// TIA Portal V21 program export: 5 tag tables, 1 data types, 6 data blocks, 4 code blocks (in call order from the OBs), 2 instance data blocks

VAR_GLOBAL   // PLC tag table "A0.300"
   tESTE_01 AT %I15.0 : Bool;
END_VAR

VAR_GLOBAL   // PLC tag table "Cabinet_Config"
   M_Power_line_3_4_Available AT %M100.0 : Bool;
   M_Power_line_5_6_Available AT %M100.1 : Bool;
   M_Safety_zone_3_4_Available AT %M101.0 : Bool;
   M_Safety_zone_5_6_Available AT %M101.1 : Bool;
   M_Safety_zone_7_8_Available AT %M101.2 : Bool;
   M_Fast_doors_Enabled AT %M102.0 : Bool;
   M_Wrapping_machine_Enabled AT %M102.1 : Bool;
   M_CabinetNumberOutOfRange AT %M110.0 : Bool;
   M_HWCombiNumberOutOfRange AT %M110.1 : Bool;
END_VAR
VAR_GLOBAL CONSTANT   // user constants
   K_MaxCabinetNumber : UInt := 10;   // Max. number of C0 cabinets allowed
   K_MaxHWCombiNumber : UInt := 16;   // Max. number of defined PLC hardware combinations
END_VAR

VAR_GLOBAL   // PLC tag table "Cabinet_Management"
   M_Power_cabinet AT %M2.0 : Bool;
   M_Power_L1 AT %M3.0 : Bool;
   M_Power_L2 AT %M3.1 : Bool;
   M_Power_L3 AT %M3.2 : Bool;
   M_Power_L4 AT %M3.3 : Bool;
   M_Power_L5 AT %M3.4 : Bool;
   M_Power_L6 AT %M3.5 : Bool;
   M_Buzzer AT %M4.0 : Bool;
   M_NF_Cabinet_fault AT %M5.0 : Bool;
   M_Cabinet_fault AT %M5.1 : Bool;
   M_Rearm_Power_Cabinet AT %M6.0 : Bool;
   M_Reset_safety_Z1 AT %M7.0 : Bool;
   M_Reset_safety_Z2 AT %M7.1 : Bool;
   M_Reset_safety_Z3 AT %M7.2 : Bool;
   M_Reset_safety_Z4 AT %M7.3 : Bool;
   M_Reset_safety_Z5 AT %M7.4 : Bool;
   M_Reset_safety_Z6 AT %M7.5 : Bool;
   M_Reset_safety_Z7 AT %M7.6 : Bool;
   M_Reset_safety_Z8 AT %M7.7 : Bool;
   M_Facility_OK AT %M6.7 : Bool;   // Conveyors status OK
END_VAR

VAR_GLOBAL   // PLC tag table "Default tag table"
   System_Byte AT %MB1 : Byte;
   FirstScan AT %M1.0 : Bool;
   DiagStatusUpdate AT %M1.1 : Bool;
   AlwaysTRUE AT %M1.2 : Bool;
   AlwaysFALSE AT %M1.3 : Bool;
   Clock_Byte AT %MB0 : Byte;
   Clock_10Hz AT %M0.0 : Bool;
   Clock_5Hz AT %M0.1 : Bool;
   "Clock_2.5Hz" AT %M0.2 : Bool;
   Clock_2Hz AT %M0.3 : Bool;
   "Clock_1.25Hz" AT %M0.4 : Bool;
   Clock_1Hz AT %M0.5 : Bool;
   "Clock_0.625Hz" AT %M0.6 : Bool;
   "Clock_0.5Hz" AT %M0.7 : Bool;
   "+C0_K0.001" AT %I0.0 : Bool;   // Phase monitor OK
   "+C0_AUX/OK" AT %I0.1 : Bool;   // Auxiliary services protection OK
   "+C0_CAL/OK" AT %I0.2 : Bool;   // Heater protection OK
   "+C0_PE/OK" AT %I0.3 : Bool;   // Insulation monitor OK
   "+C0_Spare_101.4" AT %I0.4 : Bool;   // Spare
   "+C0_Spare_101.5" AT %I0.5 : Bool;   // Spare
   "+C0_Spare_101.6" AT %I0.6 : Bool;   // Spare
   "+C0_Spare_101.7" AT %I0.7 : Bool;   // Spare
   "+C0_S2.101" AT %I1.0 : Bool;   // Cabinet reset (power lines + emergencies)
   "+C0_S2.001" AT %I1.1 : Bool;   // Cabinet power lines deactivation
   "+C0_S2.002" AT %I1.2 : Bool;   // Acoustic warning stop
   "+C0_Spare_102.3" AT %I1.3 : Bool;   // Spare
   "+C0_IF5" AT %I1.4 : Bool;   // External machine interface 5
   "+C0_IF6" AT %I1.5 : Bool;   // External machine interface 6
   "+C0_IF7" AT %I1.6 : Bool;   // External machine interface 7
   "+C0_IF8" AT %I1.7 : Bool;   // External machine interface 8
   "+C0_F2.101" AT %I2.0 : Bool;   // 400V Power L1 protection OK
   "+C0_Q1.001" AT %I2.1 : Bool;   // Power L1 is active
   "+C0_1SE1" AT %I2.2 : Bool;   // Emergency stop 1 Z1 OK
   "+C0_1SE2" AT %I2.3 : Bool;   // Emergency stop 2 Z1 OK
   "+C0_F2.102" AT %I2.4 : Bool;   // 400V Power L2 protection OK
   "+C0_Q1.002" AT %I2.5 : Bool;   // Power L2 is active
   "+C0_2SE1" AT %I2.6 : Bool;   // Emergency stop 1 Z2 OK
   "+C0_2SE2" AT %I2.7 : Bool;   // Emergency stop 2 Z2 OK
   "+C0_F2.103" AT %I3.0 : Bool;   // 400V Power L3 protection OK
   "+C0_Q1.003" AT %I3.1 : Bool;   // Power L3 is active
   "+C0_3SE1" AT %I3.2 : Bool;   // Emergency stop 1 Z3 OK
   "+C0_3SE2" AT %I3.3 : Bool;   // Emergency stop 2 Z3 OK
   "+C0_F2.104" AT %I3.4 : Bool;   // 400V Power L4 protection OK
   "+C0_Q1.004" AT %I3.5 : Bool;   // Power L4 is active
   "+C0_4SE1" AT %I3.6 : Bool;   // Emergency stop 1 Z4 OK
   "+C0_4SE2" AT %I3.7 : Bool;   // Emergency stop 2 Z4 OK
   "+C0_F2.105" AT %I4.0 : Bool;   // 400V Power L5 protection OK
   "+C0_Q1.005" AT %I4.1 : Bool;   // Power L5 is active
   "+C0_5SE1" AT %I4.2 : Bool;   // Emergency stop 1 Z5 OK
   "+C0_5SE2" AT %I4.3 : Bool;   // Emergency stop 2 Z5 OK
   "+C0_F2.106" AT %I4.4 : Bool;   // 400V Power L6 protection OK
   "+C0_Q1.006" AT %I4.5 : Bool;   // Power L6 is active
   "+C0_6SE1" AT %I4.6 : Bool;   // Emergency stop 1 Z6 OK
   "+C0_6SE2" AT %I4.7 : Bool;   // Emergency stop 2 Z6 OK
   "+C0_Spare_106.1" AT %I5.1 : Bool;   // Spare
   "+C0_7SE1" AT %I5.2 : Bool;   // Emergency stop 1 Z7 OK
   "+C0_7SE2" AT %I5.3 : Bool;   // Emergency stop 2 Z7 OK
   "+C0_Spare_106.4" AT %I5.4 : Bool;   // Spare
   "+C0_Spare_106.5" AT %I5.5 : Bool;   // Spare
   "+C0_8SE1" AT %I5.6 : Bool;   // Emergency stop 1 Z8 OK
   "+C0_8SE2" AT %I5.7 : Bool;   // Emergency stop 2 Z8 OK
   "+C0_F0.199 -F2.199" AT %I6.0 : Bool;   // Wrapping machine protection OK
   "+C0_ENF1" AT %I6.1 : Bool;   // Wrapping machine is ready
   "+C0_ENF2" AT %I6.2 : Bool;   // Wrapping machine entry consent
   "+C0_ENF3" AT %I6.3 : Bool;   // Wrapping machine completed process
   "+C0_Spare_107.4" AT %I6.4 : Bool;   // Spare
   "+C0_Spare_107.5" AT %I6.5 : Bool;   // Spare
   "+C0_Spare_107.6" AT %I6.6 : Bool;   // Spare
   "+C0_Spare_107.7" AT %I6.7 : Bool;   // Spare
   "+C0_F0.190+" AT %I7.0 : Bool;   // Fast doors protection OK
   "+C0_1PR1" AT %I7.1 : Bool;   // Fast door 1 is open
   "+C0_1PR2" AT %I7.2 : Bool;   // Fast door 1 is closed
   "+C0_2PR1" AT %I7.3 : Bool;   // Fast door 2 is open
   "+C0_2PR2" AT %I7.4 : Bool;   // Fast door 2 is closed
   "+C0_3PR1" AT %I7.5 : Bool;   // Fast door 3 is open
   "+C0_3PR2" AT %I7.6 : Bool;   // Fast door 3 is closed
   "+C0_Spare_108.7" AT %I7.7 : Bool;   // Spare
   "+C0_Buzzer" AT %Q0.0 : Bool;   // Beacon buzzer
   "+C0_Beacon_Green" AT %Q0.1 : Bool;   // Beacon green lamp
   "+C0_Beacon_Red" AT %Q0.2 : Bool;   // Beacon red lamp
   "+C0_Spare_151.3" AT %Q0.3 : Bool;   // Spare
   "+C0_PEM" AT %Q0.4 : Bool;   // Cabinet emergency stop is active
   "+C0_RE" AT %Q0.5 : Bool;   // Cabinet power lines are active
   "+C0_Spare_151.6" AT %Q0.6 : Bool;   // Spare
   "+C0_Spare_151.7" AT %Q0.7 : Bool;   // Spare
   "+C0_K1.007" AT %Q1.0 : Bool;   // External machine interface 1
   "+C0_K1.008" AT %Q1.1 : Bool;   // External machine interface 2
   "+C0_K1.009" AT %Q1.2 : Bool;   // External machine interface 3
   "+C0_K1.010" AT %Q1.3 : Bool;   // External machine interface 4
   "+C0_Spare_152.4" AT %Q1.4 : Bool;   // Spare
   "+C0_Spare_152.5" AT %Q1.5 : Bool;   // Spare
   "+C0_Spare_152.6" AT %Q1.6 : Bool;   // Spare
   "+C0_Spare_152.7" AT %Q1.7 : Bool;   // Spare
   "+C0_K1.001" AT %Q2.0 : Bool;   // 400V Power L1 activation
   "+C0_K1.002" AT %Q2.1 : Bool;   // 400V Power L2 activation
   "+C0_K1.003" AT %Q2.2 : Bool;   // 400V Power L3 activation
   "+C0_K1.004" AT %Q2.3 : Bool;   // 400V Power L4 activation
   "+C0_K1.005" AT %Q2.4 : Bool;   // 400V Power L5 activation
   "+C0_K1.006" AT %Q2.5 : Bool;   // 400V Power L6 activation
   "+C0_Spare_153.6" AT %Q2.6 : Bool;   // Spare
   "+C0_Spare_153.7" AT %Q2.7 : Bool;   // Spare
   "+C0_K1.020" AT %Q3.0 : Bool;   // Wrapping machine exit request
   "+C0_Spare_154.1" AT %Q3.1 : Bool;   // Spare
   "+C0_K1.030" AT %Q3.2 : Bool;   // Open fast door 1
   "+C0_K1.031" AT %Q3.3 : Bool;   // Close fast door 1
   "+C0_K1.032" AT %Q3.4 : Bool;   // Open fast door 2
   "+C0_K1.033" AT %Q3.5 : Bool;   // Close fast door 2
   "+C0_K1.035" AT %Q3.7 : Bool;   // Close fast door 3
   "+C0_S1.001_1" AT %I100.0 : Bool;   // Cabinet emergency stop ch1
   "+C0_Spare_201.1" AT %I100.1 : Bool;   // Spare
   "+C0_Spare_201.2" AT %I100.2 : Bool;   // Spare
   "+C0_Spare_201.3" AT %I100.3 : Bool;   // Spare
   "+C0_S1.001_2" AT %I100.4 : Bool;   // Cabinet emergency stop ch2
   "+C0_Spare_201.5" AT %I100.5 : Bool;   // Spare
   "+C0_Spare_201.6" AT %I100.6 : Bool;   // Spare
   "+C0_Spare_201.7" AT %I100.7 : Bool;   // Spare
   "+C0_1EM1" AT %I107.0 : Bool;   // Emergency stop Z1 ch1
   "+C0_2EM1" AT %I107.1 : Bool;   // Emergency stop Z2 ch1
   "+C0_K4.011-111-012-112" AT %I107.2 : Bool;   // Safety Z1 relays feedback
   "+C0_Spare_202.3" AT %I107.3 : Bool;   // Spare
   "+C0_1EM2" AT %I107.4 : Bool;   // Emergency stop Z1 ch2
   "+C0_2EM2" AT %I107.5 : Bool;   // Emergency stop Z2 ch2
   "+C0_K4.021-121-022-122" AT %I107.6 : Bool;   // Safety Z2 relays feedback
   "+C0_Spare_202.7" AT %I107.7 : Bool;   // Sapre
   "+C0_3EM1" AT %I114.0 : Bool;   // Emergency stop Z3 ch1
   "+C0_4EM1" AT %I114.1 : Bool;   // Emergency stop Z4 ch1
   "+C0_K4.031-131-032-132" AT %I114.2 : Bool;   // Safety Z3 relays feedback
   "+C0_Spare_203.3" AT %I114.3 : Bool;   // Spare
   "+C0_3EM2" AT %I114.4 : Bool;   // Emergency stop Z3 ch2
   "+C0_4EM2" AT %I114.5 : Bool;   // Emergency stop Z4 ch2
   "+C0_K4.041-141-042-142" AT %I114.6 : Bool;   // Safety Z4 relays feedback
   "+C0_Spare_203.7" AT %I114.7 : Bool;   // Spare
   "+C0_5EM1" AT %I121.0 : Bool;   // Emergency stop Z5 ch1
   "+C0_6EM1" AT %I121.1 : Bool;   // Emergency stop Z6 ch1
   "+C0_K4.051-151-052-152" AT %I121.2 : Bool;   // Safety Z5 relays feedback
   "+C0_Spare_204.3" AT %I121.3 : Bool;   // Spare
   "+C0_5EM2" AT %I121.4 : Bool;   // Emergency stop Z5 ch2
   "+C0_6EM2" AT %I121.5 : Bool;   // Emergency stop Z6 ch2
   "+C0_K4.061-161-062-162" AT %I121.6 : Bool;   // Safety Z6 relays feedback
   "+C0_Spare_204.7" AT %I121.7 : Bool;   // Spare
   "+C0_7EM1" AT %I128.0 : Bool;   // Emergency stop Z7 ch1
   "+C0_8EM1" AT %I128.1 : Bool;   // Emergency stop Z8 ch1
   "+C0_K4.071-171-072-172" AT %I128.2 : Bool;   // Safety Z7 relays feedback
   "+C0_Spare_205.3" AT %I128.3 : Bool;   // Spare
   "+C0_7EM2" AT %I128.4 : Bool;   // Emergency stop Z7 ch2
   "+C0_8EM2" AT %I128.5 : Bool;   // Emergency stop Z8 ch2
   "+C0_K4.081-181-082-182" AT %I128.6 : Bool;   // Safety Z8 relays feedback
   "+C0_Spare_205.7" AT %I128.7 : Bool;   // Spare
   "+C0_K4.011-111" AT %Q200.0 : Bool;   // Safety Z1 ch1 relay activation
   "+C0_K4.012-112" AT %Q200.1 : Bool;   // Safety Z1 ch2 relay activation
   "+C0_K4.021-121" AT %Q200.2 : Bool;   // Safety Z2 ch1 relay activation
   "+C0_K4.022-122" AT %Q200.3 : Bool;   // Safety Z2 ch2 relay activation
   "+C0_K4.031-131" AT %Q200.4 : Bool;   // Safety Z3 ch1 relay activation
   "+C0_K4.032-132" AT %Q200.5 : Bool;   // Safety Z3 ch2 relay activation
   "+C0_K4.041-141" AT %Q200.6 : Bool;   // Safety Z4 ch1 relay activation
   "+C0_K4.042-142" AT %Q200.7 : Bool;   // Safety Z4 ch2 relay activation
   "+C0_K4.051-151" AT %Q206.0 : Bool;   // Safety Z5 ch1 relay activation
   "+C0_K4.052-152" AT %Q206.1 : Bool;   // Safety Z5 ch2 relay activation
   "+C0_K4.061-161" AT %Q206.2 : Bool;   // Safety Z6 ch1 relay activation
   "+C0_K4.062-162" AT %Q206.3 : Bool;   // Safety Z6 ch2 relay activation
   "+C0_K4.071-171" AT %Q206.4 : Bool;   // Safety Z7 ch1 relay activation
   "+C0_K4.072-172" AT %Q206.5 : Bool;   // Safety Z7 ch2 relay activation
   "+C0_K4.081-181" AT %Q206.6 : Bool;   // Safety Z8 ch1 relay activation
   "+C0_K4.082-182" AT %Q206.7 : Bool;   // Safety Z8 ch2 relay activation
   "+C0_A0.101" AT %IB0 : Byte;
   "+C0_A0.102" AT %IB1 : Byte;
   "+C0_A0.103" AT %IB2 : Byte;
   "+C0_A0.104" AT %IB3 : Byte;
   "+C0_A0.105" AT %IB4 : Byte;
   "+C0_A0.106" AT %IB5 : Byte;
   "+C0_A0.107" AT %IB6 : Byte;
   "+C0_A0.108" AT %IB7 : Byte;
   "+C0_Spare_106.0" AT %I5.0 : Bool;   // Spare
   "+C0_K1.034" AT %Q3.6 : Bool;   // Open fast door 3
   RONDI_PEM_20260514 AT %M650.0 : Bool;   // VARIABLE DE PUESTA EN MARCHA
END_VAR

VAR_GLOBAL   // PLC tag table "Process_Data"
   IB_Byte0 AT %IB400 : Byte;
   IB_Byte1 AT %IB401 : Byte;
   OB_Byte0 AT %QB400 : Byte;
   OB_Byte1 AT %QB401 : Byte;
   OB_Byte2 AT %QB402 : Byte;
   OB_Byte3 AT %QB403 : Byte;
   OB_Byte4 AT %QB404 : Byte;
   OB_Byte5 AT %QB405 : Byte;
   OB_Byte6 AT %QB406 : Byte;
   OB_Byte7 AT %QB407 : Byte;
   OB_Byte8 AT %QB408 : Byte;
   OB_Byte9 AT %QB409 : Byte;
   OB_Byte10 AT %QB410 : Byte;
   IB_Byte2 AT %IB402 : Byte;
   IB_Byte3 AT %IB403 : Byte;
   OB_Byte11 AT %QB411 : Byte;
END_VAR

TYPE "TypeC0"
   STRUCT
      Heated_Lines_Enabled : Bool;   // true = Heated line/s are enabled
      Insulation_Monitor_Enabled : Bool;   // true = Insulation monitor is enabled
      Power_L2_Disabled : Bool;   // true = Power L2 is disabled
      Power_L4_Disabled : Bool;   // true = Power L4 is disabled
      Power_L6_Disabled : Bool;   // true = Power L6 is disabled
      Safety_Z2_Disabled : Bool;   // true = Safety Z2 is disabled
      Safety_Z4_Disabled : Bool;   // true = Safety Z4 is disabled
      Safety_Z6_Disabled : Bool;   // true = Safety Z6 is disabled
      Safety_Z8_Disabled : Bool;   // true = Safety Z8 is disabled
      HWCombiNumber : Int;   // PLC hardware combination number
   END_STRUCT;
END_TYPE

DATA_BLOCK "HWData"   // DB3
{ S7_Optimized_Access := 'TRUE' }
// stored: AutoNumber false, MemoryReserve 0
   VAR
      CombiNumber : Int := 0;   // Number according to PLC hardware combination
      ConfigSlots : Array[1.."K_MaxHWCombiNumber"] of "LCC_typeCPUET200SP";   // Slots configurations for all PLC hardware combinations
      CPUET200SP_StatusID : USInt;
      CPUET200SP_Status : DWord;
      CPUET200SP_Config { S7_SetPoint := 'True'} : "LCC_typeCPUET200SP";   // Slots configuration for selected hardware combination
   END_VAR
BEGIN
   ConfigSlots[1].slots[4].actSlotNumber := 132;
   ConfigSlots[1].slots[5].actSlotNumber := 133;
   ConfigSlots[1].slots[6].actSlotNumber := 134;
   ConfigSlots[1].slots[7].actSlotNumber := 7;
   ConfigSlots[1].slots[8].actSlotNumber := 136;
   ConfigSlots[1].slots[9].actSlotNumber := 9;
   ConfigSlots[1].slots[10].actSlotNumber := 10;
   ConfigSlots[1].slots[11].actSlotNumber := 11;
   ConfigSlots[1].slots[12..16].actSlotNumber := 0;
   ConfigSlots[1].slots[17].actSlotNumber := 12;
   ConfigSlots[1].slots[18].actSlotNumber := 13;
   ConfigSlots[1].slots[19].actSlotNumber := 14;
   ConfigSlots[1].slots[20].actSlotNumber := 0;
   ConfigSlots[1].slots[21].actSlotNumber := 15;
   ConfigSlots[2].slots[4].actSlotNumber := 132;
   ConfigSlots[2].slots[5].actSlotNumber := 133;
   ConfigSlots[2].slots[6].actSlotNumber := 134;
   ConfigSlots[2].slots[7].actSlotNumber := 7;
   ConfigSlots[2].slots[8].actSlotNumber := 136;
   ConfigSlots[2].slots[9].actSlotNumber := 9;
   ConfigSlots[2].slots[10].actSlotNumber := 10;
   ConfigSlots[2].slots[11].actSlotNumber := 11;
   ConfigSlots[2].slots[12..14].actSlotNumber := 0;
   ConfigSlots[2].slots[15].actSlotNumber := 12;
   ConfigSlots[2].slots[16].actSlotNumber := 0;
   ConfigSlots[2].slots[17].actSlotNumber := 13;
   ConfigSlots[2].slots[18].actSlotNumber := 14;
   ConfigSlots[2].slots[19].actSlotNumber := 15;
   ConfigSlots[2].slots[20].actSlotNumber := 16;
   ConfigSlots[2].slots[21].actSlotNumber := 17;
   ConfigSlots[3].slots[4].actSlotNumber := 132;
   ConfigSlots[3].slots[5].actSlotNumber := 133;
   ConfigSlots[3].slots[6].actSlotNumber := 134;
   ConfigSlots[3].slots[7].actSlotNumber := 7;
   ConfigSlots[3].slots[8].actSlotNumber := 136;
   ConfigSlots[3].slots[9].actSlotNumber := 9;
   ConfigSlots[3].slots[10].actSlotNumber := 10;
   ConfigSlots[3].slots[11].actSlotNumber := 11;
   ConfigSlots[3].slots[12..15].actSlotNumber := 0;
   ConfigSlots[3].slots[16].actSlotNumber := 12;
   ConfigSlots[3].slots[17].actSlotNumber := 13;
   ConfigSlots[3].slots[18].actSlotNumber := 14;
   ConfigSlots[3].slots[19].actSlotNumber := 15;
   ConfigSlots[3].slots[20].actSlotNumber := 16;
   ConfigSlots[3].slots[21].actSlotNumber := 17;
   ConfigSlots[4].slots[4].actSlotNumber := 132;
   ConfigSlots[4].slots[5].actSlotNumber := 133;
   ConfigSlots[4].slots[6].actSlotNumber := 134;
   ConfigSlots[4].slots[7].actSlotNumber := 7;
   ConfigSlots[4].slots[8].actSlotNumber := 136;
   ConfigSlots[4].slots[9].actSlotNumber := 9;
   ConfigSlots[4].slots[10].actSlotNumber := 10;
   ConfigSlots[4].slots[11].actSlotNumber := 11;
   ConfigSlots[4].slots[12..14].actSlotNumber := 0;
   ConfigSlots[4].slots[15].actSlotNumber := 12;
   ConfigSlots[4].slots[16].actSlotNumber := 13;
   ConfigSlots[4].slots[17].actSlotNumber := 14;
   ConfigSlots[4].slots[18].actSlotNumber := 15;
   ConfigSlots[4].slots[19].actSlotNumber := 16;
   ConfigSlots[4].slots[20].actSlotNumber := 17;
   ConfigSlots[4].slots[21].actSlotNumber := 18;
   ConfigSlots[5].slots[5].actSlotNumber := 133;
   ConfigSlots[5].slots[6].actSlotNumber := 134;
   ConfigSlots[5].slots[7].actSlotNumber := 7;
   ConfigSlots[5].slots[8].actSlotNumber := 136;
   ConfigSlots[5].slots[9].actSlotNumber := 9;
   ConfigSlots[5].slots[10].actSlotNumber := 10;
   ConfigSlots[5].slots[11].actSlotNumber := 11;
   ConfigSlots[5].slots[12].actSlotNumber := 12;
   ConfigSlots[5].slots[13..16].actSlotNumber := 0;
   ConfigSlots[5].slots[17].actSlotNumber := 13;
   ConfigSlots[5].slots[18].actSlotNumber := 14;
   ConfigSlots[5].slots[19].actSlotNumber := 15;
   ConfigSlots[5].slots[20].actSlotNumber := 0;
   ConfigSlots[5].slots[21].actSlotNumber := 16;
   ConfigSlots[6].slots[5].actSlotNumber := 133;
   ConfigSlots[6].slots[6].actSlotNumber := 134;
   ConfigSlots[6].slots[7].actSlotNumber := 7;
   ConfigSlots[6].slots[8].actSlotNumber := 136;
   ConfigSlots[6].slots[9].actSlotNumber := 9;
   ConfigSlots[6].slots[10].actSlotNumber := 10;
   ConfigSlots[6].slots[11].actSlotNumber := 11;
   ConfigSlots[6].slots[12].actSlotNumber := 12;
   ConfigSlots[6].slots[13..14].actSlotNumber := 0;
   ConfigSlots[6].slots[15].actSlotNumber := 13;
   ConfigSlots[6].slots[16].actSlotNumber := 0;
   ConfigSlots[6].slots[17].actSlotNumber := 14;
   ConfigSlots[6].slots[18].actSlotNumber := 15;
   ConfigSlots[6].slots[19].actSlotNumber := 16;
   ConfigSlots[6].slots[20].actSlotNumber := 17;
   ConfigSlots[6].slots[21].actSlotNumber := 18;
   ConfigSlots[7].slots[5].actSlotNumber := 133;
   ConfigSlots[7].slots[6].actSlotNumber := 134;
   ConfigSlots[7].slots[7].actSlotNumber := 7;
   ConfigSlots[7].slots[8].actSlotNumber := 136;
   ConfigSlots[7].slots[9].actSlotNumber := 9;
   ConfigSlots[7].slots[10].actSlotNumber := 10;
   ConfigSlots[7].slots[11].actSlotNumber := 11;
   ConfigSlots[7].slots[12].actSlotNumber := 12;
   ConfigSlots[7].slots[13..15].actSlotNumber := 0;
   ConfigSlots[7].slots[16].actSlotNumber := 13;
   ConfigSlots[7].slots[17].actSlotNumber := 14;
   ConfigSlots[7].slots[18].actSlotNumber := 15;
   ConfigSlots[7].slots[19].actSlotNumber := 16;
   ConfigSlots[7].slots[20].actSlotNumber := 17;
   ConfigSlots[7].slots[21].actSlotNumber := 18;
   ConfigSlots[8].slots[5].actSlotNumber := 133;
   ConfigSlots[8].slots[6].actSlotNumber := 134;
   ConfigSlots[8].slots[7].actSlotNumber := 7;
   ConfigSlots[8].slots[8].actSlotNumber := 136;
   ConfigSlots[8].slots[9].actSlotNumber := 9;
   ConfigSlots[8].slots[10].actSlotNumber := 10;
   ConfigSlots[8].slots[11].actSlotNumber := 11;
   ConfigSlots[8].slots[12].actSlotNumber := 12;
   ConfigSlots[8].slots[13..14].actSlotNumber := 0;
   ConfigSlots[8].slots[15].actSlotNumber := 13;
   ConfigSlots[8].slots[16].actSlotNumber := 14;
   ConfigSlots[8].slots[17].actSlotNumber := 15;
   ConfigSlots[8].slots[18].actSlotNumber := 16;
   ConfigSlots[8].slots[19].actSlotNumber := 17;
   ConfigSlots[8].slots[20].actSlotNumber := 18;
   ConfigSlots[8].slots[21].actSlotNumber := 19;
   ConfigSlots[9].slots[6].actSlotNumber := 134;
   ConfigSlots[9].slots[7].actSlotNumber := 7;
   ConfigSlots[9].slots[8].actSlotNumber := 8;
   ConfigSlots[9].slots[9].actSlotNumber := 9;
   ConfigSlots[9].slots[10].actSlotNumber := 10;
   ConfigSlots[9].slots[11].actSlotNumber := 11;
   ConfigSlots[9].slots[12].actSlotNumber := 12;
   ConfigSlots[9].slots[13].actSlotNumber := 13;
   ConfigSlots[9].slots[14..16].actSlotNumber := 0;
   ConfigSlots[9].slots[17].actSlotNumber := 14;
   ConfigSlots[9].slots[18].actSlotNumber := 15;
   ConfigSlots[9].slots[19].actSlotNumber := 16;
   ConfigSlots[9].slots[20].actSlotNumber := 0;
   ConfigSlots[9].slots[21].actSlotNumber := 17;
   ConfigSlots[10].slots[6].actSlotNumber := 134;
   ConfigSlots[10].slots[7].actSlotNumber := 7;
   ConfigSlots[10].slots[8].actSlotNumber := 8;
   ConfigSlots[10].slots[9].actSlotNumber := 9;
   ConfigSlots[10].slots[10].actSlotNumber := 10;
   ConfigSlots[10].slots[11].actSlotNumber := 11;
   ConfigSlots[10].slots[12].actSlotNumber := 12;
   ConfigSlots[10].slots[13].actSlotNumber := 13;
   ConfigSlots[10].slots[14].actSlotNumber := 0;
   ConfigSlots[10].slots[15].actSlotNumber := 14;
   ConfigSlots[10].slots[16].actSlotNumber := 0;
   ConfigSlots[10].slots[17].actSlotNumber := 15;
   ConfigSlots[10].slots[18].actSlotNumber := 16;
   ConfigSlots[10].slots[19].actSlotNumber := 17;
   ConfigSlots[10].slots[20].actSlotNumber := 18;
   ConfigSlots[10].slots[21].actSlotNumber := 19;
   ConfigSlots[11].slots[6].actSlotNumber := 134;
   ConfigSlots[11].slots[7].actSlotNumber := 7;
   ConfigSlots[11].slots[8].actSlotNumber := 8;
   ConfigSlots[11].slots[9].actSlotNumber := 9;
   ConfigSlots[11].slots[10].actSlotNumber := 10;
   ConfigSlots[11].slots[11].actSlotNumber := 11;
   ConfigSlots[11].slots[12].actSlotNumber := 12;
   ConfigSlots[11].slots[13].actSlotNumber := 13;
   ConfigSlots[11].slots[14..15].actSlotNumber := 0;
   ConfigSlots[11].slots[16].actSlotNumber := 14;
   ConfigSlots[11].slots[17].actSlotNumber := 15;
   ConfigSlots[11].slots[18].actSlotNumber := 16;
   ConfigSlots[11].slots[19].actSlotNumber := 17;
   ConfigSlots[11].slots[20].actSlotNumber := 18;
   ConfigSlots[11].slots[21].actSlotNumber := 19;
   ConfigSlots[12].slots[6].actSlotNumber := 134;
   ConfigSlots[12].slots[7].actSlotNumber := 7;
   ConfigSlots[12].slots[8].actSlotNumber := 8;
   ConfigSlots[12].slots[9].actSlotNumber := 9;
   ConfigSlots[12].slots[10].actSlotNumber := 10;
   ConfigSlots[12].slots[11].actSlotNumber := 11;
   ConfigSlots[12].slots[12].actSlotNumber := 12;
   ConfigSlots[12].slots[13].actSlotNumber := 13;
   ConfigSlots[12].slots[14].actSlotNumber := 0;
   ConfigSlots[12].slots[15].actSlotNumber := 14;
   ConfigSlots[12].slots[16].actSlotNumber := 15;
   ConfigSlots[12].slots[17].actSlotNumber := 16;
   ConfigSlots[12].slots[18].actSlotNumber := 17;
   ConfigSlots[12].slots[19].actSlotNumber := 18;
   ConfigSlots[12].slots[20].actSlotNumber := 19;
   ConfigSlots[12].slots[21].actSlotNumber := 20;
   ConfigSlots[13].slots[8].actSlotNumber := 8;
   ConfigSlots[13].slots[9].actSlotNumber := 9;
   ConfigSlots[13].slots[10].actSlotNumber := 10;
   ConfigSlots[13].slots[11].actSlotNumber := 11;
   ConfigSlots[13].slots[12].actSlotNumber := 12;
   ConfigSlots[13].slots[13].actSlotNumber := 13;
   ConfigSlots[13].slots[14].actSlotNumber := 14;
   ConfigSlots[13].slots[15..16].actSlotNumber := 0;
   ConfigSlots[13].slots[17].actSlotNumber := 15;
   ConfigSlots[13].slots[18].actSlotNumber := 16;
   ConfigSlots[13].slots[19].actSlotNumber := 17;
   ConfigSlots[13].slots[20].actSlotNumber := 0;
   ConfigSlots[13].slots[21].actSlotNumber := 18;
   ConfigSlots[14].slots[9].actSlotNumber := 9;
   ConfigSlots[14].slots[10].actSlotNumber := 10;
   ConfigSlots[14].slots[11].actSlotNumber := 11;
   ConfigSlots[14].slots[12].actSlotNumber := 12;
   ConfigSlots[14].slots[13].actSlotNumber := 13;
   ConfigSlots[14].slots[14].actSlotNumber := 14;
   ConfigSlots[14].slots[15].actSlotNumber := 15;
   ConfigSlots[14].slots[16].actSlotNumber := 0;
   ConfigSlots[14].slots[17].actSlotNumber := 16;
   ConfigSlots[14].slots[18].actSlotNumber := 17;
   ConfigSlots[14].slots[19].actSlotNumber := 18;
   ConfigSlots[14].slots[20].actSlotNumber := 19;
   ConfigSlots[14].slots[21].actSlotNumber := 20;
   ConfigSlots[15].slots[8].actSlotNumber := 8;
   ConfigSlots[15].slots[9].actSlotNumber := 9;
   ConfigSlots[15].slots[10].actSlotNumber := 10;
   ConfigSlots[15].slots[11].actSlotNumber := 11;
   ConfigSlots[15].slots[12].actSlotNumber := 12;
   ConfigSlots[15].slots[13].actSlotNumber := 13;
   ConfigSlots[15].slots[14].actSlotNumber := 14;
   ConfigSlots[15].slots[15].actSlotNumber := 0;
   ConfigSlots[15].slots[16].actSlotNumber := 15;
   ConfigSlots[15].slots[17].actSlotNumber := 16;
   ConfigSlots[15].slots[18].actSlotNumber := 17;
   ConfigSlots[15].slots[19].actSlotNumber := 18;
   ConfigSlots[15].slots[20].actSlotNumber := 19;
   ConfigSlots[15].slots[21].actSlotNumber := 20;
   ConfigSlots[16].slots[21].actSlotNumber := 21;
   ConfigSlots[1].slots[2].slotProperty := 1;
   ConfigSlots[1].slots[4..6].slotProperty := 0;
END_DATA_BLOCK

DATA_BLOCK "C0_DATA"   // DB10
{ S7_Optimized_Access := 'TRUE' }
// stored: MemoryReserve 100
   VAR
      C0 : "TypeC0";   // Copy of the current cabinet configuration
   END_VAR
BEGIN
END_DATA_BLOCK

DATA_BLOCK "C0_ID"   // DB9
{ S7_Optimized_Access := 'TRUE' }
// stored: MemoryReserve 100
   VAR
      CabinetNumber : Int := 1;   // Current C0 cabinet to be programmed
   END_VAR
BEGIN
END_DATA_BLOCK

DATA_BLOCK "Cabinets_Config"   // DB8
{ S7_Optimized_Access := 'TRUE' }
// stored: MemoryReserve 100
   VAR
      C0 : Array[1.."K_MaxCabinetNumber"] of "TypeC0";
   END_VAR
BEGIN
   C0[1].Power_L2_Disabled := false;
   C0[1].Power_L4_Disabled := false;
   C0[1].Safety_Z2_Disabled := true;
   C0[1].Safety_Z4_Disabled := false;
   C0[1].HWCombiNumber := 1;
   C0[2].HWCombiNumber := 3;
   C0[3..4].HWCombiNumber := 1;
END_DATA_BLOCK

DATA_BLOCK "LCC_ConfigDevice_DB"
{ S7_Optimized_Access := 'TRUE' }
AUTHOR : SIOS
FAMILY : LCC
VERSION : 1.0
NON_RETAIN
"LCC_ConfigDevice"

BEGIN

END_DATA_BLOCK

DATA_BLOCK "Buzzer timer"
{InstructionName := 'IEC_TIMER';
 LibVersion := '1.0';
 S7_Optimized_Access := 'TRUE' }
AUTHOR : Simatic
FAMILY : IEC
NAME : IEC_TMR
VERSION : 1.0
NON_RETAIN
IEC_TIMER

BEGIN

END_DATA_BLOCK

ORGANIZATION_BLOCK "Main"   // OB1, LAD, ProgramCycle
TITLE = "Main Program Sweep (Cycle)"
{ S7_Optimized_Access := 'TRUE' }
// stored: SetENOAutomatically false
   VAR_INPUT
      Initial_Call : Bool;   // Initial call of this OB
      Remanence : Bool;   // =True, if remanent data are available
   END_VAR
BEGIN

REGION Network 1: Cabinet management
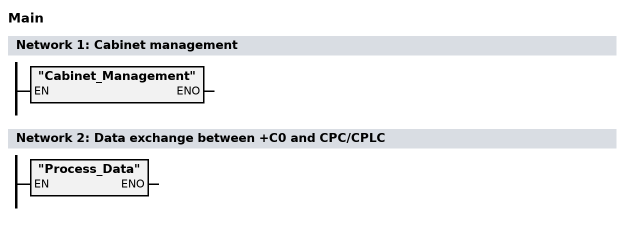
   RUNG wire#powerrail
      "Cabinet_Management"()
   END_RUNG
   // the same network as SCL:
   "Cabinet_Management"();
END_REGION

REGION Network 2: Data exchange between +C0 and CPC/CPLC
   RUNG wire#powerrail
      "Process_Data"()
   END_RUNG
   // the same network as SCL:
   "Process_Data"();
END_REGION
END_ORGANIZATION_BLOCK

FUNCTION "Cabinet_Management" : Void   // FC1, LAD
{ S7_Optimized_Access := 'TRUE' }
// stored: SetENOAutomatically false
   VAR_TEMP
      Phase_monitor_OK : Bool;
      Auxiliary_sevices_OK : Bool;
      "400V_protections_OK" : Bool;
      "400V_power_lines_activated" : Bool;
      Aux_emergencies : Bool;
      Emergencies_OK : Bool;
      Aux_cabinet_OK : Bool;
      Cabinet_OK : Bool;
      Heater_OK : Bool;
      Insulation_Monitor_OK : Bool;
      Power_wrapping_machine_OK : Bool;
      Power_fast_doors_OK : Bool;
      Facility_fault : Bool;
      Summary_fault : Bool;
   END_VAR
   VAR_TEMP   // added for the SCL form of the ladder/FBD networks
      _w1 : Bool;
      _w2 : Bool;
   END_VAR
BEGIN

REGION Network 1: Cabinet power control
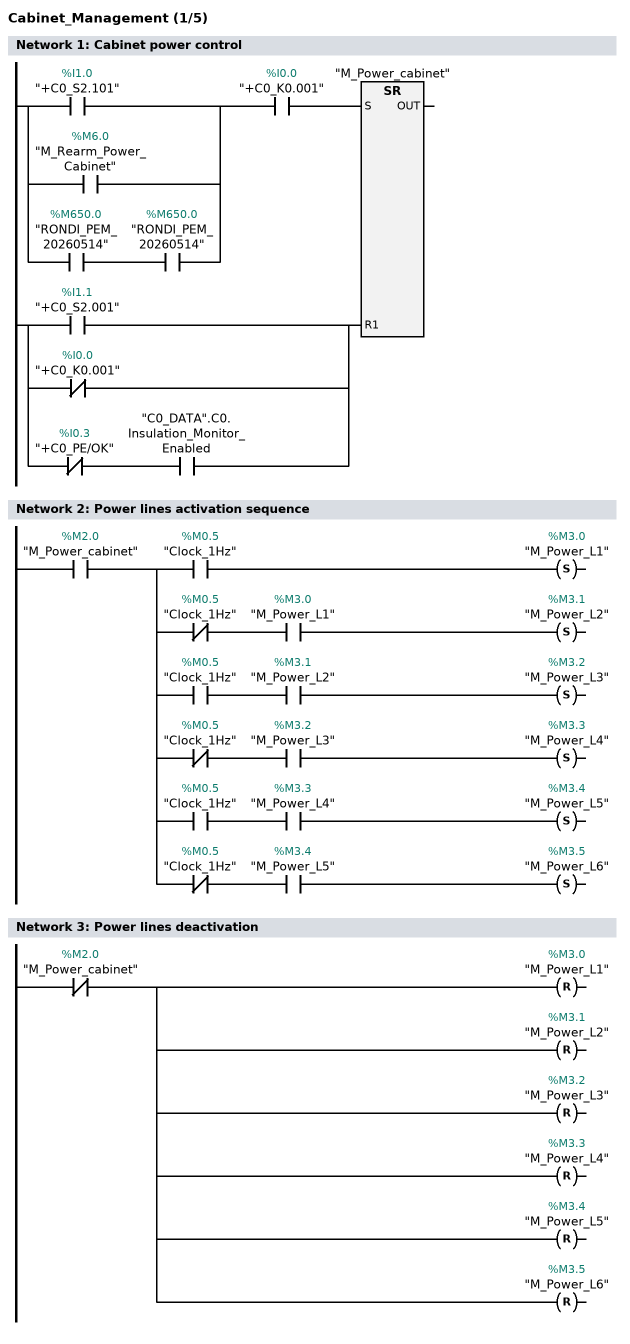
   RUNG wire#powerrail
      Contact( "+C0_S2.101" )
      wire#w1
      Contact( "+C0_K0.001" )
      S_SR(operand := "M_Power_cabinet", r1 := wire#w2)
   END_RUNG
   RUNG wire#powerrail
      Contact( "M_Rearm_Power_Cabinet" )
   END_RUNG wire#w1
   RUNG wire#powerrail
      Contact( "RONDI_PEM_20260514" )
      Contact( "RONDI_PEM_20260514" )
   END_RUNG wire#w1
   RUNG wire#powerrail
      Contact( "+C0_S2.001" )
   END_RUNG wire#w2
   RUNG wire#powerrail
      I_Contact( "+C0_K0.001" )
   END_RUNG wire#w2
   RUNG wire#powerrail
      I_Contact( "+C0_PE/OK" )
      Contact( "C0_DATA".C0.Insulation_Monitor_Enabled )
   END_RUNG wire#w2
   // the same network as SCL:
   IF ("+C0_S2.101" OR "M_Rearm_Power_Cabinet" OR ("RONDI_PEM_20260514" AND "RONDI_PEM_20260514")) AND "+C0_K0.001" THEN
       "M_Power_cabinet" := TRUE;   // SR flip-flop
   END_IF;
   IF "+C0_S2.001" OR NOT "+C0_K0.001" OR (NOT "+C0_PE/OK" AND "C0_DATA".C0.Insulation_Monitor_Enabled) THEN
       "M_Power_cabinet" := FALSE;
   END_IF;
END_REGION

REGION Network 2: Power lines activation sequence
   RUNG wire#powerrail
      Contact( "M_Power_cabinet" )
      wire#w1
      Contact( "Clock_1Hz" )
      S_Coil( "M_Power_L1" )
   END_RUNG
   RUNG wire#w1
      I_Contact( "Clock_1Hz" )
      Contact( "M_Power_L1" )
      S_Coil( "M_Power_L2" )
   END_RUNG
   RUNG wire#w1
      Contact( "Clock_1Hz" )
      Contact( "M_Power_L2" )
      S_Coil( "M_Power_L3" )
   END_RUNG
   RUNG wire#w1
      I_Contact( "Clock_1Hz" )
      Contact( "M_Power_L3" )
      S_Coil( "M_Power_L4" )
   END_RUNG
   RUNG wire#w1
      Contact( "Clock_1Hz" )
      Contact( "M_Power_L4" )
      S_Coil( "M_Power_L5" )
   END_RUNG
   RUNG wire#w1
      I_Contact( "Clock_1Hz" )
      Contact( "M_Power_L5" )
      S_Coil( "M_Power_L6" )
   END_RUNG
   // the same network as SCL:
   IF "M_Power_cabinet" AND "Clock_1Hz" THEN "M_Power_L1" := TRUE; END_IF;
   IF "M_Power_cabinet" AND NOT "Clock_1Hz" AND "M_Power_L1" THEN "M_Power_L2" := TRUE; END_IF;
   IF "M_Power_cabinet" AND "Clock_1Hz" AND "M_Power_L2" THEN "M_Power_L3" := TRUE; END_IF;
   IF "M_Power_cabinet" AND NOT "Clock_1Hz" AND "M_Power_L3" THEN "M_Power_L4" := TRUE; END_IF;
   IF "M_Power_cabinet" AND "Clock_1Hz" AND "M_Power_L4" THEN "M_Power_L5" := TRUE; END_IF;
   IF "M_Power_cabinet" AND NOT "Clock_1Hz" AND "M_Power_L5" THEN "M_Power_L6" := TRUE; END_IF;
END_REGION

REGION Network 3: Power lines deactivation
   RUNG wire#powerrail
      I_Contact( "M_Power_cabinet" )
      wire#w1
      R_Coil( "M_Power_L1" )
   END_RUNG
   RUNG wire#w1
      R_Coil( "M_Power_L2" )
   END_RUNG
   RUNG wire#w1
      R_Coil( "M_Power_L3" )
   END_RUNG
   RUNG wire#w1
      R_Coil( "M_Power_L4" )
   END_RUNG
   RUNG wire#w1
      R_Coil( "M_Power_L5" )
   END_RUNG
   RUNG wire#w1
      R_Coil( "M_Power_L6" )
   END_RUNG
   // the same network as SCL:
   IF NOT "M_Power_cabinet" THEN
       "M_Power_L1" := FALSE;
       "M_Power_L2" := FALSE;
       "M_Power_L3" := FALSE;
       "M_Power_L4" := FALSE;
       "M_Power_L5" := FALSE;
       "M_Power_L6" := FALSE;
   END_IF;
END_REGION

REGION Network 4: Power lines outputs
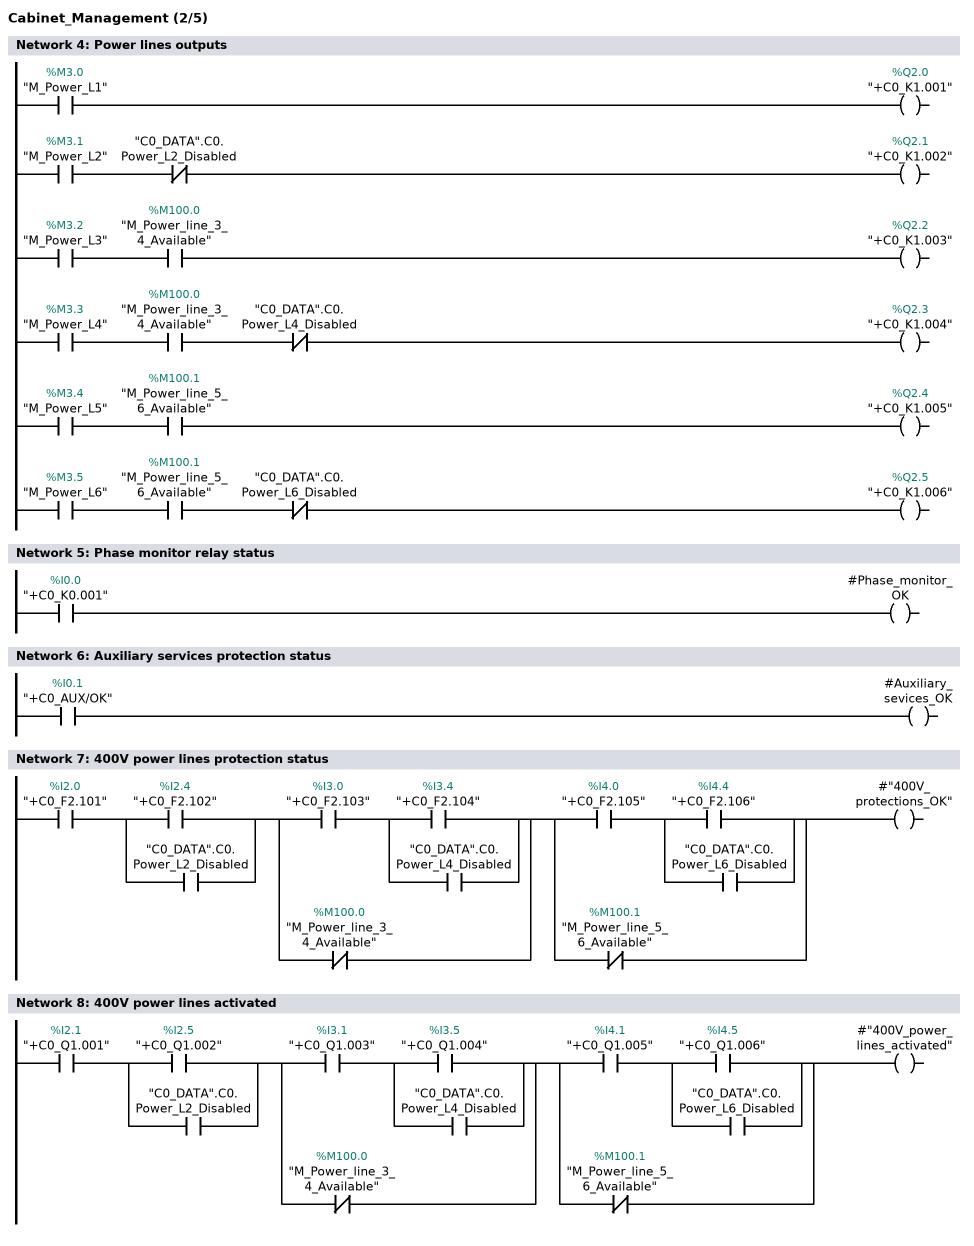
   RUNG wire#powerrail
      Contact( "M_Power_L1" )
      Coil( "+C0_K1.001" )
   END_RUNG
   RUNG wire#powerrail
      Contact( "M_Power_L2" )
      I_Contact( "C0_DATA".C0.Power_L2_Disabled )
      Coil( "+C0_K1.002" )
   END_RUNG
   RUNG wire#powerrail
      Contact( "M_Power_L3" )
      Contact( "M_Power_line_3_4_Available" )
      Coil( "+C0_K1.003" )
   END_RUNG
   RUNG wire#powerrail
      Contact( "M_Power_L4" )
      Contact( "M_Power_line_3_4_Available" )
      I_Contact( "C0_DATA".C0.Power_L4_Disabled )
      Coil( "+C0_K1.004" )
   END_RUNG
   RUNG wire#powerrail
      Contact( "M_Power_L5" )
      Contact( "M_Power_line_5_6_Available" )
      Coil( "+C0_K1.005" )
   END_RUNG
   RUNG wire#powerrail
      Contact( "M_Power_L6" )
      Contact( "M_Power_line_5_6_Available" )
      I_Contact( "C0_DATA".C0.Power_L6_Disabled )
      Coil( "+C0_K1.006" )
   END_RUNG
   // the same network as SCL:
   "+C0_K1.001" := "M_Power_L1";
   "+C0_K1.002" := "M_Power_L2" AND NOT "C0_DATA".C0.Power_L2_Disabled;
   "+C0_K1.003" := "M_Power_L3" AND "M_Power_line_3_4_Available";
   "+C0_K1.004" := "M_Power_L4" AND "M_Power_line_3_4_Available" AND NOT "C0_DATA".C0.Power_L4_Disabled;
   "+C0_K1.005" := "M_Power_L5" AND "M_Power_line_5_6_Available";
   "+C0_K1.006" := "M_Power_L6" AND "M_Power_line_5_6_Available" AND NOT "C0_DATA".C0.Power_L6_Disabled;
END_REGION

REGION Network 5: Phase monitor relay status
   RUNG wire#powerrail
      Contact( "+C0_K0.001" )
      Coil( #Phase_monitor_OK )
   END_RUNG
   // the same network as SCL:
   #Phase_monitor_OK := "+C0_K0.001";
END_REGION

REGION Network 6: Auxiliary services protection status
   RUNG wire#powerrail
      Contact( "+C0_AUX/OK" )
      Coil( #Auxiliary_sevices_OK )
   END_RUNG
   // the same network as SCL:
   #Auxiliary_sevices_OK := "+C0_AUX/OK";
END_REGION

REGION Network 7: 400V power lines protection status
   RUNG wire#powerrail
      Contact( "+C0_F2.101" )
      wire#w1
      Contact( "+C0_F2.102" )
      wire#w2
      Contact( "+C0_F2.103" )
      wire#w3
      Contact( "+C0_F2.104" )
      wire#w4
      Contact( "+C0_F2.105" )
      wire#w5
      Contact( "+C0_F2.106" )
      wire#w6
      Coil( #"400V_protections_OK" )
   END_RUNG
   RUNG wire#w1
      Contact( "C0_DATA".C0.Power_L2_Disabled )
   END_RUNG wire#w2
   RUNG wire#w3
      Contact( "C0_DATA".C0.Power_L4_Disabled )
   END_RUNG wire#w4
   RUNG wire#w2
      I_Contact( "M_Power_line_3_4_Available" )
   END_RUNG wire#w4
   RUNG wire#w5
      Contact( "C0_DATA".C0.Power_L6_Disabled )
   END_RUNG wire#w6
   RUNG wire#w4
      I_Contact( "M_Power_line_5_6_Available" )
   END_RUNG wire#w6
   // the same network as SCL:
   #"400V_protections_OK" := "+C0_F2.101" AND ("+C0_F2.102" OR "C0_DATA".C0.Power_L2_Disabled) AND (("+C0_F2.103" AND ("+C0_F2.104" OR "C0_DATA".C0.Power_L4_Disabled)) OR NOT "M_Power_line_3_4_Available") AND (("+C0_F2.105" AND ("+C0_F2.106" OR "C0_DATA".C0.Power_L6_Disabled)) OR NOT "M_Power_line_5_6_Available");
END_REGION

REGION Network 8: 400V power lines activated
   RUNG wire#powerrail
      Contact( "+C0_Q1.001" )
      wire#w1
      Contact( "+C0_Q1.002" )
      wire#w2
      Contact( "+C0_Q1.003" )
      wire#w3
      Contact( "+C0_Q1.004" )
      wire#w4
      Contact( "+C0_Q1.005" )
      wire#w5
      Contact( "+C0_Q1.006" )
      wire#w6
      Coil( #"400V_power_lines_activated" )
   END_RUNG
   RUNG wire#w1
      Contact( "C0_DATA".C0.Power_L2_Disabled )
   END_RUNG wire#w2
   RUNG wire#w3
      Contact( "C0_DATA".C0.Power_L4_Disabled )
   END_RUNG wire#w4
   RUNG wire#w2
      I_Contact( "M_Power_line_3_4_Available" )
   END_RUNG wire#w4
   RUNG wire#w5
      Contact( "C0_DATA".C0.Power_L6_Disabled )
   END_RUNG wire#w6
   RUNG wire#w4
      I_Contact( "M_Power_line_5_6_Available" )
   END_RUNG wire#w6
   // the same network as SCL:
   #"400V_power_lines_activated" := "+C0_Q1.001" AND ("+C0_Q1.002" OR "C0_DATA".C0.Power_L2_Disabled) AND (("+C0_Q1.003" AND ("+C0_Q1.004" OR "C0_DATA".C0.Power_L4_Disabled)) OR NOT "M_Power_line_3_4_Available") AND (("+C0_Q1.005" AND ("+C0_Q1.006" OR "C0_DATA".C0.Power_L6_Disabled)) OR NOT "M_Power_line_5_6_Available");
END_REGION

REGION Network 9: Emergency stops + Safety lines status
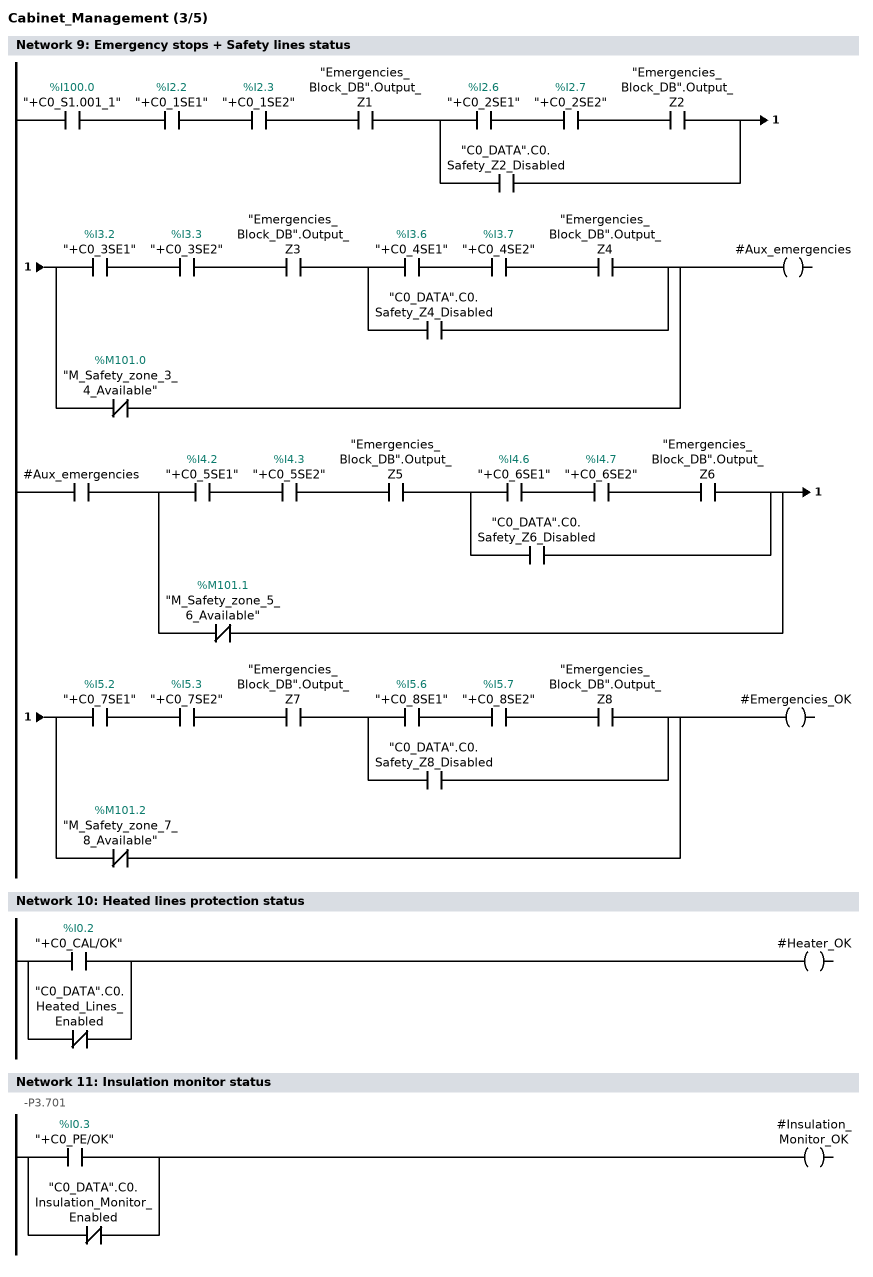
   RUNG wire#powerrail
      Contact( "+C0_S1.001_1" )
      Contact( "+C0_1SE1" )
      Contact( "+C0_1SE2" )
      Contact( "Emergencies_Block_DB".Output_Z1 )
      wire#w1
      Contact( "+C0_2SE1" )
      Contact( "+C0_2SE2" )
      Contact( "Emergencies_Block_DB".Output_Z2 )
      wire#w2
      Contact( "+C0_3SE1" )
      Contact( "+C0_3SE2" )
      Contact( "Emergencies_Block_DB".Output_Z3 )
      wire#w3
      Contact( "+C0_4SE1" )
      Contact( "+C0_4SE2" )
      Contact( "Emergencies_Block_DB".Output_Z4 )
      wire#w4
      Coil( #Aux_emergencies )
   END_RUNG
   RUNG wire#w1
      Contact( "C0_DATA".C0.Safety_Z2_Disabled )
   END_RUNG wire#w2
   RUNG wire#w3
      Contact( "C0_DATA".C0.Safety_Z4_Disabled )
   END_RUNG wire#w4
   RUNG wire#w2
      I_Contact( "M_Safety_zone_3_4_Available" )
   END_RUNG wire#w4
   RUNG wire#powerrail
      Contact( #Aux_emergencies )
      wire#w5
      Contact( "+C0_5SE1" )
      Contact( "+C0_5SE2" )
      Contact( "Emergencies_Block_DB".Output_Z5 )
      wire#w6
      Contact( "+C0_6SE1" )
      Contact( "+C0_6SE2" )
      Contact( "Emergencies_Block_DB".Output_Z6 )
      wire#w7
      Contact( "+C0_7SE1" )
      Contact( "+C0_7SE2" )
      Contact( "Emergencies_Block_DB".Output_Z7 )
      wire#w8
      Contact( "+C0_8SE1" )
      Contact( "+C0_8SE2" )
      Contact( "Emergencies_Block_DB".Output_Z8 )
      wire#w9
      Coil( #Emergencies_OK )
   END_RUNG
   RUNG wire#w6
      Contact( "C0_DATA".C0.Safety_Z6_Disabled )
   END_RUNG wire#w7
   RUNG wire#w5
      I_Contact( "M_Safety_zone_5_6_Available" )
   END_RUNG wire#w7
   RUNG wire#w8
      Contact( "C0_DATA".C0.Safety_Z8_Disabled )
   END_RUNG wire#w9
   RUNG wire#w7
      I_Contact( "M_Safety_zone_7_8_Available" )
   END_RUNG wire#w9
   // the same network as SCL:
   #Aux_emergencies := "+C0_S1.001_1" AND "+C0_1SE1" AND "+C0_1SE2" AND "Emergencies_Block_DB".Output_Z1 AND (("+C0_2SE1" AND "+C0_2SE2" AND "Emergencies_Block_DB".Output_Z2) OR "C0_DATA".C0.Safety_Z2_Disabled) AND (("+C0_3SE1" AND "+C0_3SE2" AND "Emergencies_Block_DB".Output_Z3 AND (("+C0_4SE1" AND "+C0_4SE2" AND "Emergencies_Block_DB".Output_Z4) OR "C0_DATA".C0.Safety_Z4_Disabled)) OR NOT "M_Safety_zone_3_4_Available");
   #Emergencies_OK := #Aux_emergencies AND (("+C0_5SE1" AND "+C0_5SE2" AND "Emergencies_Block_DB".Output_Z5 AND (("+C0_6SE1" AND "+C0_6SE2" AND "Emergencies_Block_DB".Output_Z6) OR "C0_DATA".C0.Safety_Z6_Disabled)) OR NOT "M_Safety_zone_5_6_Available") AND (("+C0_7SE1" AND "+C0_7SE2" AND "Emergencies_Block_DB".Output_Z7 AND (("+C0_8SE1" AND "+C0_8SE2" AND "Emergencies_Block_DB".Output_Z8) OR "C0_DATA".C0.Safety_Z8_Disabled)) OR NOT "M_Safety_zone_7_8_Available");
END_REGION

REGION Network 10: Heated lines protection status
   RUNG wire#powerrail
      Contact( "+C0_CAL/OK" )
      wire#w1
      Coil( #Heater_OK )
   END_RUNG
   RUNG wire#powerrail
      I_Contact( "C0_DATA".C0.Heated_Lines_Enabled )
   END_RUNG wire#w1
   // the same network as SCL:
   #Heater_OK := "+C0_CAL/OK" OR NOT "C0_DATA".C0.Heated_Lines_Enabled;
END_REGION

REGION Network 11: Insulation monitor status
   // -P3.701
   RUNG wire#powerrail
      Contact( "+C0_PE/OK" )
      wire#w1
      Coil( #Insulation_Monitor_OK )
   END_RUNG
   RUNG wire#powerrail
      I_Contact( "C0_DATA".C0.Insulation_Monitor_Enabled )
   END_RUNG wire#w1
   // the same network as SCL:
   #Insulation_Monitor_OK := "+C0_PE/OK" OR NOT "C0_DATA".C0.Insulation_Monitor_Enabled;
END_REGION

REGION Network 12: Wrapping machine protection status
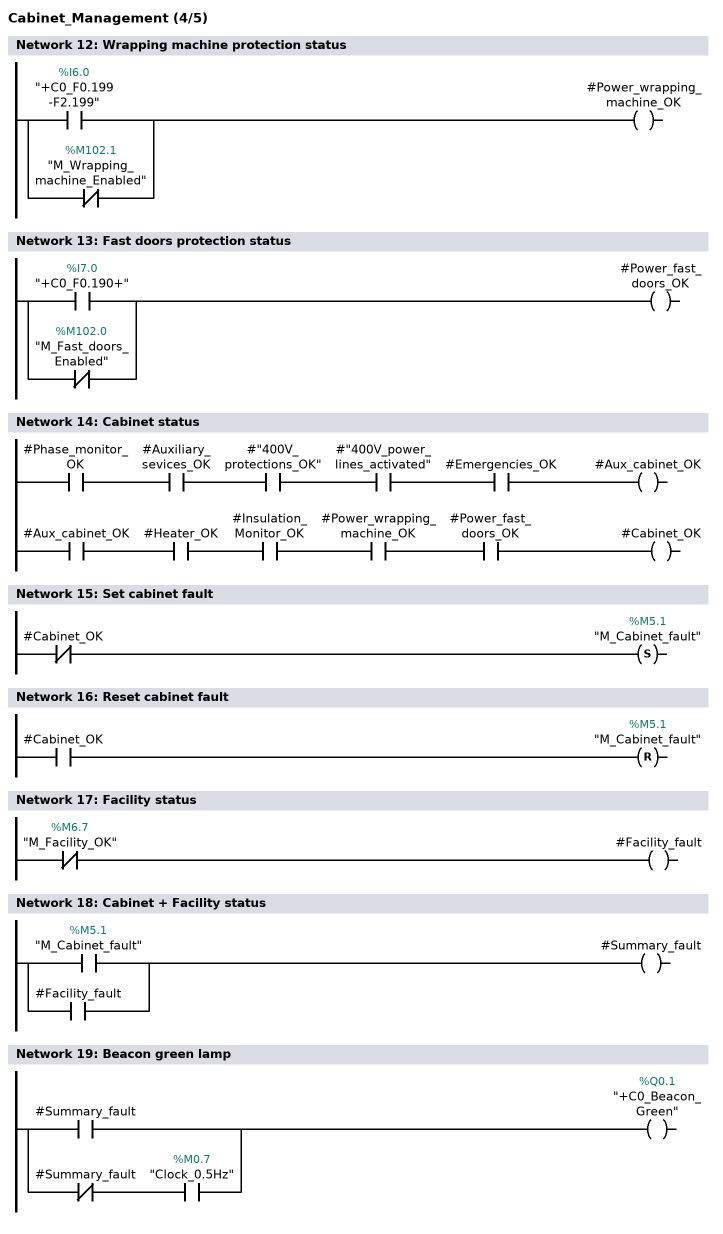
   RUNG wire#powerrail
      Contact( "+C0_F0.199 -F2.199" )
      wire#w1
      Coil( #Power_wrapping_machine_OK )
   END_RUNG
   RUNG wire#powerrail
      I_Contact( "M_Wrapping_machine_Enabled" )
   END_RUNG wire#w1
   // the same network as SCL:
   #Power_wrapping_machine_OK := "+C0_F0.199 -F2.199" OR NOT "M_Wrapping_machine_Enabled";
END_REGION

REGION Network 13: Fast doors protection status
   RUNG wire#powerrail
      Contact( "+C0_F0.190+" )
      wire#w1
      Coil( #Power_fast_doors_OK )
   END_RUNG
   RUNG wire#powerrail
      I_Contact( "M_Fast_doors_Enabled" )
   END_RUNG wire#w1
   // the same network as SCL:
   #Power_fast_doors_OK := "+C0_F0.190+" OR NOT "M_Fast_doors_Enabled";
END_REGION

REGION Network 14: Cabinet status
   RUNG wire#powerrail
      Contact( #Phase_monitor_OK )
      Contact( #Auxiliary_sevices_OK )
      Contact( #"400V_protections_OK" )
      Contact( #"400V_power_lines_activated" )
      Contact( #Emergencies_OK )
      Coil( #Aux_cabinet_OK )
   END_RUNG
   RUNG wire#powerrail
      Contact( #Aux_cabinet_OK )
      Contact( #Heater_OK )
      Contact( #Insulation_Monitor_OK )
      Contact( #Power_wrapping_machine_OK )
      Contact( #Power_fast_doors_OK )
      Coil( #Cabinet_OK )
   END_RUNG
   // the same network as SCL:
   #Aux_cabinet_OK := #Phase_monitor_OK AND #Auxiliary_sevices_OK AND #"400V_protections_OK" AND #"400V_power_lines_activated" AND #Emergencies_OK;
   #Cabinet_OK := #Aux_cabinet_OK AND #Heater_OK AND #Insulation_Monitor_OK AND #Power_wrapping_machine_OK AND #Power_fast_doors_OK;
END_REGION

REGION Network 15: Set cabinet fault
   RUNG wire#powerrail
      I_Contact( #Cabinet_OK )
      S_Coil( "M_Cabinet_fault" )
   END_RUNG
   // the same network as SCL:
   IF NOT #Cabinet_OK THEN "M_Cabinet_fault" := TRUE; END_IF;
END_REGION

REGION Network 16: Reset cabinet fault
   RUNG wire#powerrail
      Contact( #Cabinet_OK )
      R_Coil( "M_Cabinet_fault" )
   END_RUNG
   // the same network as SCL:
   IF #Cabinet_OK THEN "M_Cabinet_fault" := FALSE; END_IF;
END_REGION

REGION Network 17: Facility status
   RUNG wire#powerrail
      I_Contact( "M_Facility_OK" )
      Coil( #Facility_fault )
   END_RUNG
   // the same network as SCL:
   #Facility_fault := NOT "M_Facility_OK";
END_REGION

REGION Network 18: Cabinet + Facility status
   RUNG wire#powerrail
      Contact( "M_Cabinet_fault" )
      wire#w1
      Coil( #Summary_fault )
   END_RUNG
   RUNG wire#powerrail
      Contact( #Facility_fault )
   END_RUNG wire#w1
   // the same network as SCL:
   #Summary_fault := "M_Cabinet_fault" OR #Facility_fault;
END_REGION

REGION Network 19: Beacon green lamp
   RUNG wire#powerrail
      Contact( #Summary_fault )
      wire#w1
      Coil( "+C0_Beacon_Green" )
   END_RUNG
   RUNG wire#powerrail
      I_Contact( #Summary_fault )
      Contact( "Clock_0.5Hz" )
   END_RUNG wire#w1
   // the same network as SCL:
   "+C0_Beacon_Green" := #Summary_fault OR (NOT #Summary_fault AND "Clock_0.5Hz");
END_REGION

REGION Network 20: Beacon red lamp
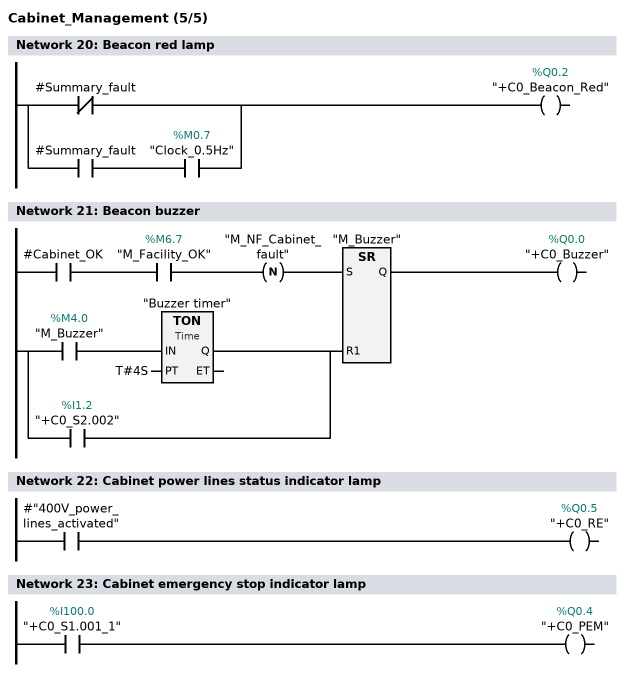
   RUNG wire#powerrail
      I_Contact( #Summary_fault )
      wire#w1
      Coil( "+C0_Beacon_Red" )
   END_RUNG
   RUNG wire#powerrail
      Contact( #Summary_fault )
      Contact( "Clock_0.5Hz" )
   END_RUNG wire#w1
   // the same network as SCL:
   "+C0_Beacon_Red" := NOT #Summary_fault OR (#Summary_fault AND "Clock_0.5Hz");
END_REGION

REGION Network 21: Beacon buzzer
   RUNG wire#powerrail
      Contact( #Cabinet_OK )
      Contact( "M_Facility_OK" )
      N_Trig( "M_NF_Cabinet_fault" )
      S_SR(operand := "M_Buzzer", r1 := wire#w1)
      Coil( "+C0_Buzzer" )
   END_RUNG
   RUNG wire#powerrail
      Contact( "M_Buzzer" )
      { S7_Templates := "time_type := Time" } "Buzzer timer".TON(pt := T#4S, et =>)
   END_RUNG wire#w1
   RUNG wire#powerrail
      Contact( "+C0_S2.002" )
   END_RUNG wire#w1
   // the same network as SCL:
   #_w1 := #Cabinet_OK AND "M_Facility_OK";
   #_w2 := NOT #_w1 AND "M_NF_Cabinet_fault";   // falling edge
   "M_NF_Cabinet_fault" := #_w1;
   "Buzzer timer".TON(IN := "M_Buzzer", PT := T#4S);
   IF #_w2 THEN
       "M_Buzzer" := TRUE;   // SR flip-flop
   END_IF;
   IF "Buzzer timer".Q OR "+C0_S2.002" THEN "M_Buzzer" := FALSE; END_IF;
   "+C0_Buzzer" := "M_Buzzer";
END_REGION

REGION Network 22: Cabinet power lines status indicator lamp
   RUNG wire#powerrail
      Contact( #"400V_power_lines_activated" )
      Coil( "+C0_RE" )
   END_RUNG
   // the same network as SCL:
   "+C0_RE" := #"400V_power_lines_activated";
END_REGION

REGION Network 23: Cabinet emergency stop indicator lamp
   RUNG wire#powerrail
      Contact( "+C0_S1.001_1" )
      Coil( "+C0_PEM" )
   END_RUNG
   // the same network as SCL:
   "+C0_PEM" := "+C0_S1.001_1";
END_REGION
END_FUNCTION

FUNCTION "Process_Data" : Void   // FC4, LAD
TITLE = PLC < - > CPC/CPLC data exchange
{ S7_Optimized_Access := 'TRUE' }
// Inputs:      Galileo -> PLC
// Outputs:  PLC -> Galileo
// stored: AutoNumber false, SetENOAutomatically false
   VAR_TEMP
      input : Byte;
   END_VAR
BEGIN

REGION Network 1: Input Byte 0 Rearm power C0 cabinet + Facility status
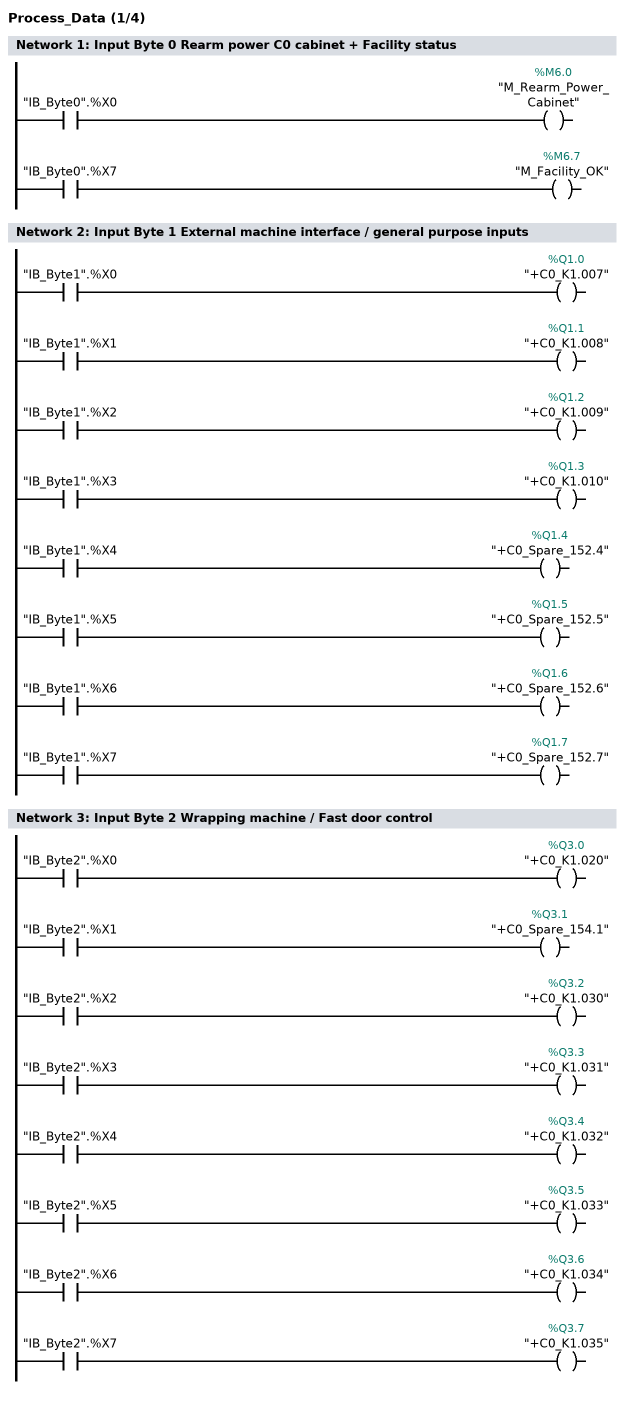
   RUNG wire#powerrail
      Contact( "IB_Byte0".%X0 )
      Coil( "M_Rearm_Power_Cabinet" )
   END_RUNG
   RUNG wire#powerrail
      Contact( "IB_Byte0".%X7 )
      Coil( "M_Facility_OK" )
   END_RUNG
   // the same network as SCL:
   "M_Rearm_Power_Cabinet" := "IB_Byte0".%X0;
   "M_Facility_OK" := "IB_Byte0".%X7;
END_REGION

REGION Network 2: Input Byte 1 External machine interface / general purpose inputs
   RUNG wire#powerrail
      Contact( "IB_Byte1".%X0 )
      Coil( "+C0_K1.007" )
   END_RUNG
   RUNG wire#powerrail
      Contact( "IB_Byte1".%X1 )
      Coil( "+C0_K1.008" )
   END_RUNG
   RUNG wire#powerrail
      Contact( "IB_Byte1".%X2 )
      Coil( "+C0_K1.009" )
   END_RUNG
   RUNG wire#powerrail
      Contact( "IB_Byte1".%X3 )
      Coil( "+C0_K1.010" )
   END_RUNG
   RUNG wire#powerrail
      Contact( "IB_Byte1".%X4 )
      Coil( "+C0_Spare_152.4" )
   END_RUNG
   RUNG wire#powerrail
      Contact( "IB_Byte1".%X5 )
      Coil( "+C0_Spare_152.5" )
   END_RUNG
   RUNG wire#powerrail
      Contact( "IB_Byte1".%X6 )
      Coil( "+C0_Spare_152.6" )
   END_RUNG
   RUNG wire#powerrail
      Contact( "IB_Byte1".%X7 )
      Coil( "+C0_Spare_152.7" )
   END_RUNG
   // the same network as SCL:
   "+C0_K1.007" := "IB_Byte1".%X0;
   "+C0_K1.008" := "IB_Byte1".%X1;
   "+C0_K1.009" := "IB_Byte1".%X2;
   "+C0_K1.010" := "IB_Byte1".%X3;
   "+C0_Spare_152.4" := "IB_Byte1".%X4;
   "+C0_Spare_152.5" := "IB_Byte1".%X5;
   "+C0_Spare_152.6" := "IB_Byte1".%X6;
   "+C0_Spare_152.7" := "IB_Byte1".%X7;
END_REGION

REGION Network 3: Input Byte 2 Wrapping machine / Fast door control
   RUNG wire#powerrail
      Contact( "IB_Byte2".%X0 )
      Coil( "+C0_K1.020" )
   END_RUNG
   RUNG wire#powerrail
      Contact( "IB_Byte2".%X1 )
      Coil( "+C0_Spare_154.1" )
   END_RUNG
   RUNG wire#powerrail
      Contact( "IB_Byte2".%X2 )
      Coil( "+C0_K1.030" )
   END_RUNG
   RUNG wire#powerrail
      Contact( "IB_Byte2".%X3 )
      Coil( "+C0_K1.031" )
   END_RUNG
   RUNG wire#powerrail
      Contact( "IB_Byte2".%X4 )
      Coil( "+C0_K1.032" )
   END_RUNG
   RUNG wire#powerrail
      Contact( "IB_Byte2".%X5 )
      Coil( "+C0_K1.033" )
   END_RUNG
   RUNG wire#powerrail
      Contact( "IB_Byte2".%X6 )
      Coil( "+C0_K1.034" )
   END_RUNG
   RUNG wire#powerrail
      Contact( "IB_Byte2".%X7 )
      Coil( "+C0_K1.035" )
   END_RUNG
   // the same network as SCL:
   "+C0_K1.020" := "IB_Byte2".%X0;
   "+C0_Spare_154.1" := "IB_Byte2".%X1;
   "+C0_K1.030" := "IB_Byte2".%X2;
   "+C0_K1.031" := "IB_Byte2".%X3;
   "+C0_K1.032" := "IB_Byte2".%X4;
   "+C0_K1.033" := "IB_Byte2".%X5;
   "+C0_K1.034" := "IB_Byte2".%X6;
   "+C0_K1.035" := "IB_Byte2".%X7;
END_REGION

REGION Network 4: Input Byte 3 Reset of safety zones
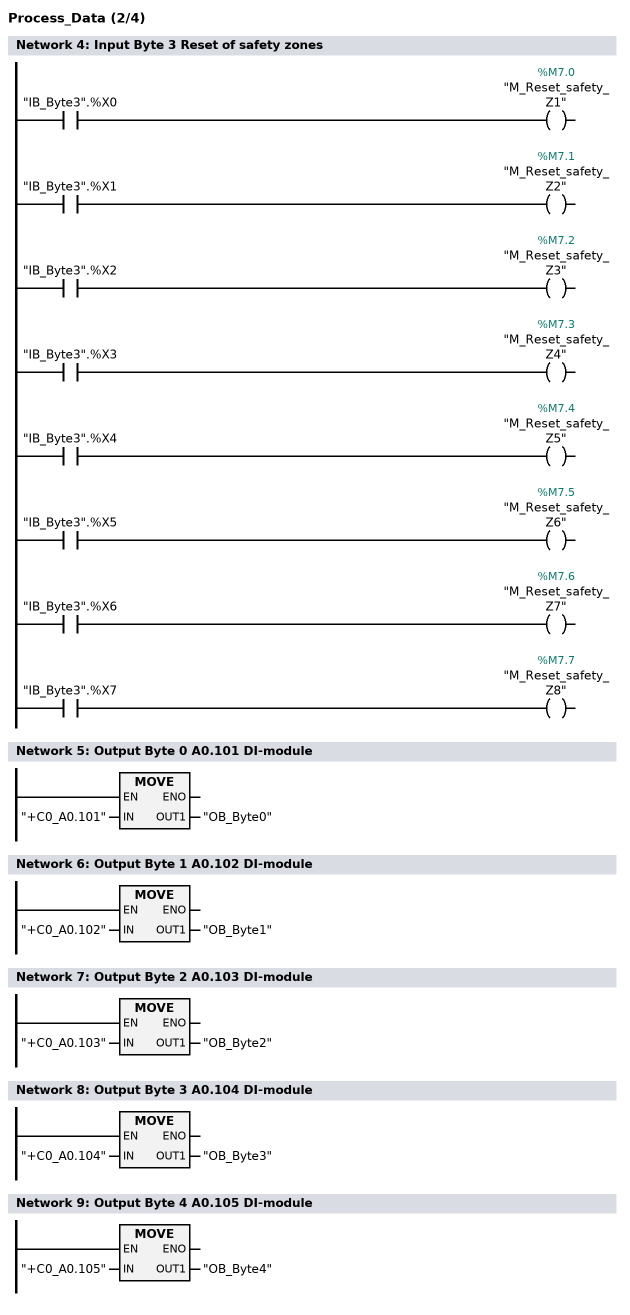
   RUNG wire#powerrail
      Contact( "IB_Byte3".%X0 )
      Coil( "M_Reset_safety_Z1" )
   END_RUNG
   RUNG wire#powerrail
      Contact( "IB_Byte3".%X1 )
      Coil( "M_Reset_safety_Z2" )
   END_RUNG
   RUNG wire#powerrail
      Contact( "IB_Byte3".%X2 )
      Coil( "M_Reset_safety_Z3" )
   END_RUNG
   RUNG wire#powerrail
      Contact( "IB_Byte3".%X3 )
      Coil( "M_Reset_safety_Z4" )
   END_RUNG
   RUNG wire#powerrail
      Contact( "IB_Byte3".%X4 )
      Coil( "M_Reset_safety_Z5" )
   END_RUNG
   RUNG wire#powerrail
      Contact( "IB_Byte3".%X5 )
      Coil( "M_Reset_safety_Z6" )
   END_RUNG
   RUNG wire#powerrail
      Contact( "IB_Byte3".%X6 )
      Coil( "M_Reset_safety_Z7" )
   END_RUNG
   RUNG wire#powerrail
      Contact( "IB_Byte3".%X7 )
      Coil( "M_Reset_safety_Z8" )
   END_RUNG
   // the same network as SCL:
   "M_Reset_safety_Z1" := "IB_Byte3".%X0;
   "M_Reset_safety_Z2" := "IB_Byte3".%X1;
   "M_Reset_safety_Z3" := "IB_Byte3".%X2;
   "M_Reset_safety_Z4" := "IB_Byte3".%X3;
   "M_Reset_safety_Z5" := "IB_Byte3".%X4;
   "M_Reset_safety_Z6" := "IB_Byte3".%X5;
   "M_Reset_safety_Z7" := "IB_Byte3".%X6;
   "M_Reset_safety_Z8" := "IB_Byte3".%X7;
END_REGION

REGION Network 5: Output Byte 0 A0.101 DI-module
   RUNG wire#powerrail
      Move(in := "+C0_A0.101", out1 => "OB_Byte0")
   END_RUNG
   // the same network as SCL:
   "OB_Byte0" := "+C0_A0.101";
END_REGION

REGION Network 6: Output Byte 1 A0.102 DI-module
   RUNG wire#powerrail
      Move(in := "+C0_A0.102", out1 => "OB_Byte1")
   END_RUNG
   // the same network as SCL:
   "OB_Byte1" := "+C0_A0.102";
END_REGION

REGION Network 7: Output Byte 2 A0.103 DI-module
   RUNG wire#powerrail
      Move(in := "+C0_A0.103", out1 => "OB_Byte2")
   END_RUNG
   // the same network as SCL:
   "OB_Byte2" := "+C0_A0.103";
END_REGION

REGION Network 8: Output Byte 3 A0.104 DI-module
   RUNG wire#powerrail
      Move(in := "+C0_A0.104", out1 => "OB_Byte3")
   END_RUNG
   // the same network as SCL:
   "OB_Byte3" := "+C0_A0.104";
END_REGION

REGION Network 9: Output Byte 4 A0.105 DI-module
   RUNG wire#powerrail
      Move(in := "+C0_A0.105", out1 => "OB_Byte4")
   END_RUNG
   // the same network as SCL:
   "OB_Byte4" := "+C0_A0.105";
END_REGION

REGION Network 10: Output Byte 5 A0.106 DI-module
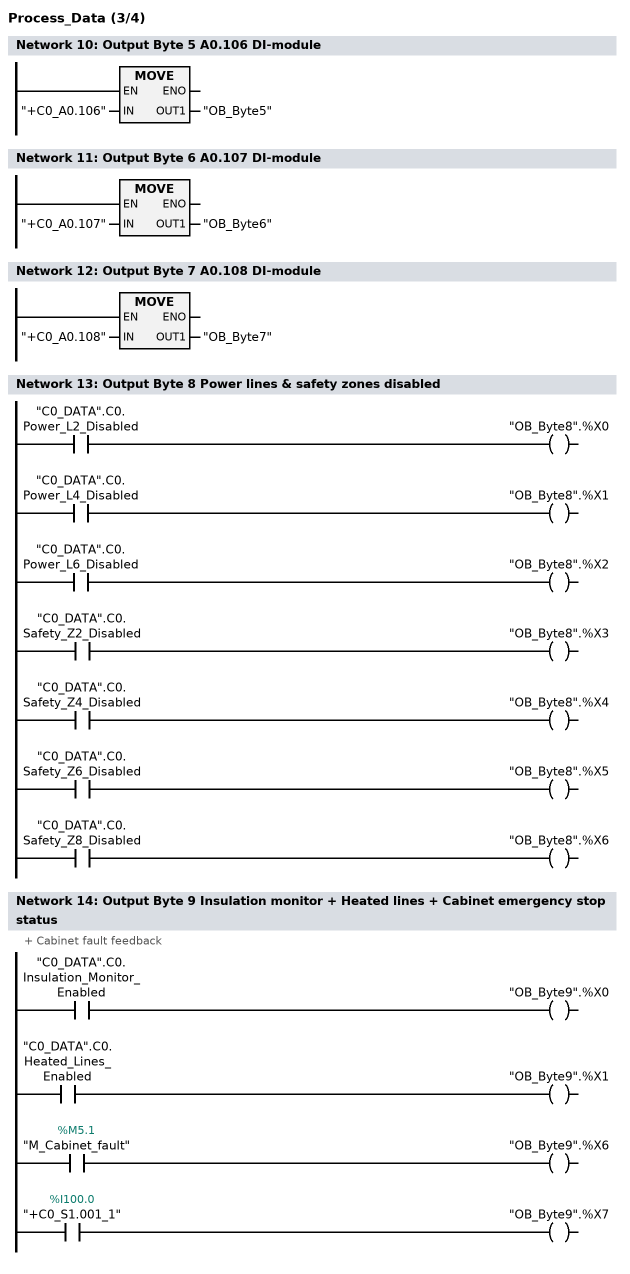
   RUNG wire#powerrail
      Move(in := "+C0_A0.106", out1 => "OB_Byte5")
   END_RUNG
   // the same network as SCL:
   "OB_Byte5" := "+C0_A0.106";
END_REGION

REGION Network 11: Output Byte 6 A0.107 DI-module
   RUNG wire#powerrail
      Move(in := "+C0_A0.107", out1 => "OB_Byte6")
   END_RUNG
   // the same network as SCL:
   "OB_Byte6" := "+C0_A0.107";
END_REGION

REGION Network 12: Output Byte 7 A0.108 DI-module
   RUNG wire#powerrail
      Move(in := "+C0_A0.108", out1 => "OB_Byte7")
   END_RUNG
   // the same network as SCL:
   "OB_Byte7" := "+C0_A0.108";
END_REGION

REGION Network 13: Output Byte 8 Power lines & safety zones disabled
   RUNG wire#powerrail
      Contact( "C0_DATA".C0.Power_L2_Disabled )
      Coil( "OB_Byte8".%X0 )
   END_RUNG
   RUNG wire#powerrail
      Contact( "C0_DATA".C0.Power_L4_Disabled )
      Coil( "OB_Byte8".%X1 )
   END_RUNG
   RUNG wire#powerrail
      Contact( "C0_DATA".C0.Power_L6_Disabled )
      Coil( "OB_Byte8".%X2 )
   END_RUNG
   RUNG wire#powerrail
      Contact( "C0_DATA".C0.Safety_Z2_Disabled )
      Coil( "OB_Byte8".%X3 )
   END_RUNG
   RUNG wire#powerrail
      Contact( "C0_DATA".C0.Safety_Z4_Disabled )
      Coil( "OB_Byte8".%X4 )
   END_RUNG
   RUNG wire#powerrail
      Contact( "C0_DATA".C0.Safety_Z6_Disabled )
      Coil( "OB_Byte8".%X5 )
   END_RUNG
   RUNG wire#powerrail
      Contact( "C0_DATA".C0.Safety_Z8_Disabled )
      Coil( "OB_Byte8".%X6 )
   END_RUNG
   // the same network as SCL:
   "OB_Byte8".%X0 := "C0_DATA".C0.Power_L2_Disabled;
   "OB_Byte8".%X1 := "C0_DATA".C0.Power_L4_Disabled;
   "OB_Byte8".%X2 := "C0_DATA".C0.Power_L6_Disabled;
   "OB_Byte8".%X3 := "C0_DATA".C0.Safety_Z2_Disabled;
   "OB_Byte8".%X4 := "C0_DATA".C0.Safety_Z4_Disabled;
   "OB_Byte8".%X5 := "C0_DATA".C0.Safety_Z6_Disabled;
   "OB_Byte8".%X6 := "C0_DATA".C0.Safety_Z8_Disabled;
END_REGION

REGION Network 14: Output Byte 9 Insulation monitor + Heated lines + Cabinet emergency stop status
   // + Cabinet fault feedback
   RUNG wire#powerrail
      Contact( "C0_DATA".C0.Insulation_Monitor_Enabled )
      Coil( "OB_Byte9".%X0 )
   END_RUNG
   RUNG wire#powerrail
      Contact( "C0_DATA".C0.Heated_Lines_Enabled )
      Coil( "OB_Byte9".%X1 )
   END_RUNG
   RUNG wire#powerrail
      Contact( "M_Cabinet_fault" )
      Coil( "OB_Byte9".%X6 )
   END_RUNG
   RUNG wire#powerrail
      Contact( "+C0_S1.001_1" )
      Coil( "OB_Byte9".%X7 )
   END_RUNG
   // the same network as SCL:
   "OB_Byte9".%X0 := "C0_DATA".C0.Insulation_Monitor_Enabled;
   "OB_Byte9".%X1 := "C0_DATA".C0.Heated_Lines_Enabled;
   "OB_Byte9".%X6 := "M_Cabinet_fault";
   "OB_Byte9".%X7 := "+C0_S1.001_1";
END_REGION

REGION Network 15: Output Byte 10 Emergency zones status
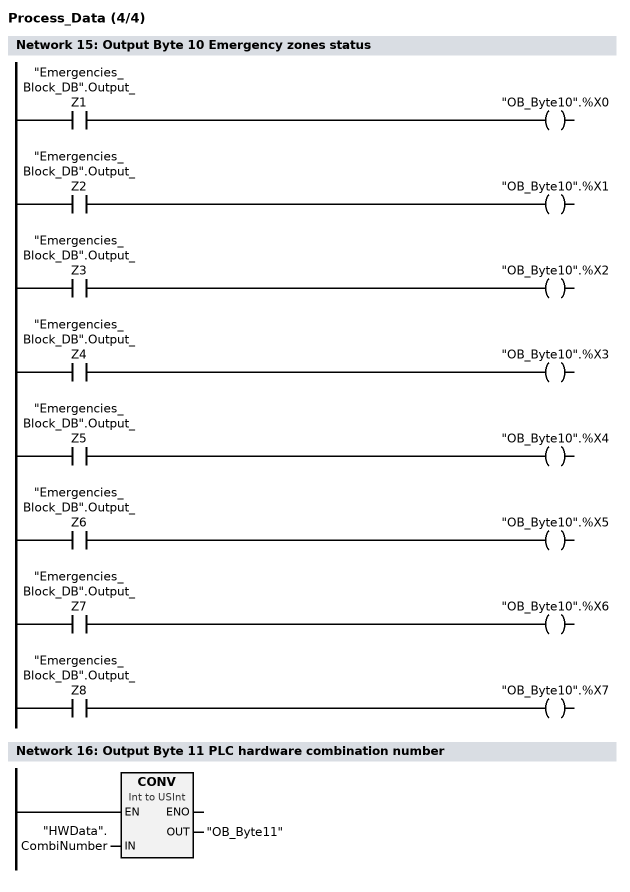
   RUNG wire#powerrail
      Contact( "Emergencies_Block_DB".Output_Z1 )
      Coil( "OB_Byte10".%X0 )
   END_RUNG
   RUNG wire#powerrail
      Contact( "Emergencies_Block_DB".Output_Z2 )
      Coil( "OB_Byte10".%X1 )
   END_RUNG
   RUNG wire#powerrail
      Contact( "Emergencies_Block_DB".Output_Z3 )
      Coil( "OB_Byte10".%X2 )
   END_RUNG
   RUNG wire#powerrail
      Contact( "Emergencies_Block_DB".Output_Z4 )
      Coil( "OB_Byte10".%X3 )
   END_RUNG
   RUNG wire#powerrail
      Contact( "Emergencies_Block_DB".Output_Z5 )
      Coil( "OB_Byte10".%X4 )
   END_RUNG
   RUNG wire#powerrail
      Contact( "Emergencies_Block_DB".Output_Z6 )
      Coil( "OB_Byte10".%X5 )
   END_RUNG
   RUNG wire#powerrail
      Contact( "Emergencies_Block_DB".Output_Z7 )
      Coil( "OB_Byte10".%X6 )
   END_RUNG
   RUNG wire#powerrail
      Contact( "Emergencies_Block_DB".Output_Z8 )
      Coil( "OB_Byte10".%X7 )
   END_RUNG
   // the same network as SCL:
   "OB_Byte10".%X0 := "Emergencies_Block_DB".Output_Z1;
   "OB_Byte10".%X1 := "Emergencies_Block_DB".Output_Z2;
   "OB_Byte10".%X2 := "Emergencies_Block_DB".Output_Z3;
   "OB_Byte10".%X3 := "Emergencies_Block_DB".Output_Z4;
   "OB_Byte10".%X4 := "Emergencies_Block_DB".Output_Z5;
   "OB_Byte10".%X5 := "Emergencies_Block_DB".Output_Z6;
   "OB_Byte10".%X6 := "Emergencies_Block_DB".Output_Z7;
   "OB_Byte10".%X7 := "Emergencies_Block_DB".Output_Z8;
END_REGION

REGION Network 16: Output Byte 11 PLC hardware combination number
   RUNG wire#powerrail
      { S7_Templates := "[SrcType := Int, DestType := USInt]" } Convert(in := "HWData".CombiNumber, out => "OB_Byte11")
   END_RUNG
   // the same network as SCL:
   "OB_Byte11" := INT_TO_USINT("HWData".CombiNumber);
END_REGION
END_FUNCTION

ORGANIZATION_BLOCK "Startup"   // OB100, LAD, Startup
TITLE = "Complete Restart"
{ S7_Optimized_Access := 'TRUE' }
// stored: SetENOAutomatically false
   VAR_INPUT
      LostRetentive : Bool;   // True if retentive data are lost
      LostRTC : Bool;   // True if date and time are lost
   END_VAR
BEGIN

REGION Network 1 (SCL): Load the selected hardware combination
   // The configuration of the slots is loaded according to the selected hardware combination
   IF (("C0_ID".CabinetNumber >= 1) AND ("C0_ID".CabinetNumber <= "K_MaxCabinetNumber")) THEN
       "HWData".CombiNumber := "Cabinets_Config".C0["C0_ID".CabinetNumber].HWCombiNumber;
       IF (("HWData".CombiNumber >= 1) AND ("HWData".CombiNumber <= "K_MaxHWCombiNumber")) THEN
           "HWData".CPUET200SP_Config := "HWData".ConfigSlots["HWData".CombiNumber];
           "C0_DATA".C0 := "Cabinets_Config".C0["C0_ID".CabinetNumber];
       ELSE
           "M_HWCombiNumberOutOfRange" := TRUE;
       END_IF;
   ELSE
       "M_CabinetNumberOutOfRange" := TRUE;
   END_IF;
END_REGION

REGION Network 2: Hardware configuration
   // For more details refer to:
   // - Configuring standard machines in TIA Portal (configuration control) Application example.
   // - Library for Configuration Control (LCC).
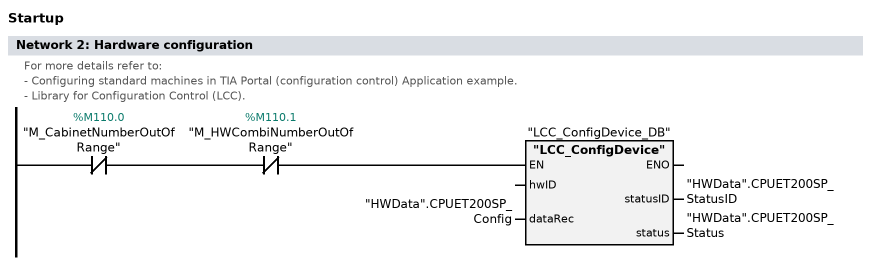
   RUNG wire#powerrail
      I_Contact( "M_CabinetNumberOutOfRange" )
      I_Contact( "M_HWCombiNumberOutOfRange" )
      "LCC_ConfigDevice_DB"(hwID :=, dataRec := "HWData".CPUET200SP_Config, statusID => "HWData".CPUET200SP_StatusID, status => "HWData".CPUET200SP_Status)
   END_RUNG
   // the same network as SCL:
   IF NOT "M_CabinetNumberOutOfRange" AND NOT "M_HWCombiNumberOutOfRange" THEN
       "LCC_ConfigDevice_DB"(dataRec := "HWData".CPUET200SP_Config,   // "LCC_ConfigDevice"
                             statusID => "HWData".CPUET200SP_StatusID,
                             status => "HWData".CPUET200SP_Status);
   END_IF;
END_REGION

REGION Network 3 (SCL): Configuration of the +C0 cabinet functionalities according to the configured hardware.
   // For all hardware combinations:
   //   - Power lines L1/L2 are always available.
   //   - Safety zones Z1/Z2 are always available.
   IF "HWData".CombiNumber > 4 THEN
       "M_Power_line_3_4_Available" := TRUE;
       "M_Safety_zone_3_4_Available" := TRUE;
   END_IF;

   IF "HWData".CombiNumber > 8 THEN
       "M_Power_line_5_6_Available" := TRUE;
       "M_Safety_zone_5_6_Available" := TRUE;
   END_IF;

   IF "HWData".CombiNumber > 12 THEN
       "M_Safety_zone_7_8_Available" := TRUE;
   END_IF;

   IF ("HWData".CombiNumber = 2 OR
       "HWData".CombiNumber = 6 OR
       "HWData".CombiNumber = 10 OR
       "HWData".CombiNumber = 14) THEN
       "M_Wrapping_machine_Enabled" := TRUE;
   END_IF;

   IF ("HWData".CombiNumber = 3 OR
       "HWData".CombiNumber = 7 OR
       "HWData".CombiNumber = 11 OR
       "HWData".CombiNumber = 15) THEN
       "M_Fast_doors_Enabled" := TRUE;
   END_IF;

   IF ("HWData".CombiNumber = 4 OR
       "HWData".CombiNumber = 8 OR
       "HWData".CombiNumber = 12 OR
       "HWData".CombiNumber = 16) THEN
       "M_Wrapping_machine_Enabled" := TRUE;
       "M_Fast_doors_Enabled" := TRUE;
   END_IF;
END_REGION
END_ORGANIZATION_BLOCK

DATA_BLOCK "LCC_ConfigDevice_DB"   // DB2
AUTHOR : SIOS
FAMILY : LCC
VERSION : 1.0
// stored: InstanceOfName LCC_ConfigDevice, InstanceOfType FB
"LCC_ConfigDevice"
   // VAR_INPUT
   //    hwID : HW_IO;
   // END_VAR
   // VAR_OUTPUT
   //    statusID : USInt;
   //    status { ExternalAccessible := 'False'; ExternalVisible := 'False'; ExternalWritable := 'False'} : DWord;
   // END_VAR
   // VAR_IN_OUT
   //    dataRec : Variant;
   // END_VAR
   // VAR
   //    statReq : Bool;
   //    instWriteRecord { ExternalAccessible := 'False'; ExternalVisible := 'False'; ExternalWritable := 'False'; S7_SetPoint := 'True'} : WRREC;
   // END_VAR
BEGIN
END_DATA_BLOCK

DATA_BLOCK "Buzzer timer"   // DB7
{ S7_Optimized_Access := 'TRUE' }
// stored: InstanceOfName IEC_TIMER, OfSystemLibElement IEC_TIMER, OfSystemLibVersion 1.0
"IEC_TIMER"
   // VAR
   //    PT : Time;
   //    ET { ExternalWritable := 'False'} : Time;
   //    IN : Bool;
   //    Q { ExternalWritable := 'False'} : Bool;
   // END_VAR
BEGIN
END_DATA_BLOCK
